   VAR_OUTPUT 
      error { ExternalAccessible := 'False'; ExternalVisible := 'False'; ExternalWritable := 'False'} : Bool;
      status { ExternalAccessible := 'False'; ExternalVisible := 'False'; ExternalWritable := 'False'} : Word;
   END_VAR

   VAR 
      statActorType { ExternalAccessible := 'False'; ExternalVisible := 'False'; ExternalWritable := 'False'} : DInt;
      statByteOffset { ExternalAccessible := 'False'; ExternalVisible := 'False'; ExternalWritable := 'False'} : Int;
      statFirstCycle { ExternalAccessible := 'False'; ExternalVisible := 'False'; ExternalWritable := 'False'} : Bool := TRUE;
      statAddressOut { ExternalAccessible := 'False'; ExternalVisible := 'False'; ExternalWritable := 'False'} : Struct
         RID { ExternalAccessible := 'False'; ExternalVisible := 'False'; ExternalWritable := 'False'} : DWord;
         AREA { ExternalAccessible := 'False'; ExternalVisible := 'False'; ExternalWritable := 'False'} : Byte;
         DB_NUMBER { ExternalAccessible := 'False'; ExternalVisible := 'False'; ExternalWritable := 'False'} : UInt;
         OFFSET { ExternalAccessible := 'False'; ExternalVisible := 'False'; ExternalWritable := 'False'} : UDInt;
      END_STRUCT;
      statNsoll { ExternalAccessible := 'False'; ExternalVisible := 'False'; ExternalWritable := 'False'} : DInt;
      statOutput { ExternalAccessible := 'False'; ExternalVisible := 'False'; ExternalWritable := 'False'} : Int;
   END_VAR

   VAR_TEMP 
      tempAttributes : Byte;
      tempDBLength : UDInt;
      tempStatus : Int;
      tempEno : Bool;
   END_VAR

   VAR CONSTANT 
      AREA_DB : Byte := 16#8B;
      STATUS_DONE : Word := 16#0000;
      STATUS_BUSY : Word := 16#7001;
      ALARM_OPTIMIZED_DB : UDInt := 9106;
      ALARM_INTERNAL : UDInt := 9201;
      ALARM_WRITE_OUTPUT : UDInt := 9401;
   END_VAR


BEGIN
	//================================================================================
	//SIEMENS AG // (c)Copyright 2019 All Rights Reserved
	//--------------------------------------------------------------------------------
	//Library:       LSimaHydTO
	//Tested with:   S7-15xx
	//Engineering:   TIA Portal  V15
	//Restrictions:  -
	//Requirements:  S7-1500 (FW 2.5)
	//Functionality: - for internal use
	//
	//--------------------------------------------------------------------------------
	//Change log table:
	//
	//Version     Date          Expert in charge    Changes applied
	//01.00.00    15.03.2018    APC_ERLF            First released version
	//================================================================================
	// Set error FALSE
	#error := FALSE;
	
	IF (#statFirstCycle)
	THEN
	  // Get adresses from TO
	  #statActorType := #axis.Actor.Type;
	  #statAddressOut.AREA := #axis.Actor.Interface.AddressOut.AREA;
	  #statAddressOut.DB_NUMBER := #axis.Actor.Interface.AddressOut.DB_NUMBER;
	  #statAddressOut.OFFSET := #axis.Actor.Interface.AddressOut.OFFSET;
	  #statAddressOut.RID := #axis.Actor.Interface.AddressOut.RID;
	  
	  IF #statActorType = 0 THEN
	    // analog
	    
	    #statByteOffset := UDINT_TO_INT(#statAddressOut.OFFSET / 8);
	  ELSIF #statActorType = 1 THEN
	    //profidrive
	    #statByteOffset := UDINT_TO_INT(#statAddressOut.OFFSET / 8) + 2;
	  END_IF;
	  
	  IF (#statAddressOut.AREA = #AREA_DB) THEN
	    #tempStatus := ATTR_DB(REQ := TRUE
	                           , DB_NUMBER := #statAddressOut.DB_NUMBER
	                           , DB_LENGTH => #tempDBLength
	                           , ATTRIB => #tempAttributes);
	    
	    IF (#tempStatus <> 0) THEN
	      // Error in reading block data
	      #error := TRUE;
	      #status := UDINT_TO_WORD(#ALARM_INTERNAL);
	      RETURN;
	      
	    ELSIF ((#tempDBLength = 0)
	      AND (#tempAttributes.%X0 = FALSE))
	    THEN
	      // Block is optimized
	      #error := TRUE;
	      #status := UDINT_TO_WORD(#ALARM_OPTIMIZED_DB);
	      RETURN;
	      
	    END_IF;
	  END_IF;
	  
	  #statFirstCycle := FALSE;
	END_IF;
	
	
	#status := #STATUS_BUSY;
	CASE #statActorType OF
	  0: // analog
	    #statOutput := LREAL_TO_INT(0.01 * #setpoint * 27648);
	    POKE(area := #statAddressOut.AREA,
	         dbNumber := #statAddressOut.DB_NUMBER,
	         byteOffset := #statByteOffset,
	         value := INT_TO_WORD(#statOutput),
	         ENO => #tempEno);
	  1: // profidrive
	    #statNsoll := LREAL_TO_DINT(LIMIT(MN := -2.0, IN := 0.01 * #setpoint, MX := 1.999999999) * 1073741824.0);
	    POKE(area := #statAddressOut.AREA,
	         dbNumber := #statAddressOut.DB_NUMBER,
	         byteOffset := #statByteOffset,
	         value := DINT_TO_DWORD(#statNsoll),
	         ENO => #tempEno);
	END_CASE;
	
	
	// Check if read worked
	IF (#tempEno = FALSE) THEN
	  #error := TRUE;
	  
	  #status := UDINT_TO_WORD(#ALARM_WRITE_OUTPUT);
	END_IF;
	
	
	
END_FUNCTION_BLOCK

FUNCTION "LSimaHydTO_GetUnitsCorrection" : LReal
{ S7_Optimized_Access := 'TRUE' }
AUTHOR : APC_ERLF
FAMILY : LSimaHydTO
VERSION : 1.0
   VAR_INPUT 
      lengthUnit : UDInt;
      velocityUnit : UDInt;
   END_VAR

   VAR_OUTPUT 
      accelFactor : LReal;
   END_VAR

   VAR_TEMP 
      tempLengthFactor : LReal;
      tempTimeFactor : LReal;
   END_VAR


BEGIN
	//================================================================================
	//SIEMENS AG // (c)Copyright 2019 All Rights Reserved
	//--------------------------------------------------------------------------------
	//Library:       LSimaHydTO
	//Tested with:   S7-15xx
	//Engineering:   TIA Portal  V15
	//Restrictions:  -
	//Requirements:  S7-1500 (FW 2.5)
	//Functionality: - for internal use
	//
	//--------------------------------------------------------------------------------
	//Change log table:
	//
	//Version     Date          Expert in charge    Changes applied
	//01.00.00    24.04.2020    APC_ERLF            First released version
	//================================================================================
	//
	
	CASE #lengthUnit OF
	    1013: //    mm
	        // get time factor
	        CASE #velocityUnit OF
	            1061, 1062: // m/s, mm/s
	                #tempTimeFactor := 1.0;
	            1524, 1525, 1527:    // mm/min, m/min, km/min
	                #tempTimeFactor := 60.0;
	            1063, 1526, 1064:    // m/h, mm/h, km/h
	                #tempTimeFactor := 3600.0;
	            ELSE
	                #tempTimeFactor := 1.0;
	        END_CASE;
	        // get length factor
	        CASE #velocityUnit OF
	            1062, 1524, 1526:  // mm/s, mm/min, mm/h
	                #tempLengthFactor := 1.0;
	                #accelFactor := 1.0;
	            1061, 1525, 1063:  // m/s, m/min, m/h
	                #tempLengthFactor := 1000.0;
	                #accelFactor := 0.001;
	            1064, 1527: //   km/h, km/min
	                #tempLengthFactor := 1000000.0;
	                #accelFactor := 0.001;
	            ELSE
	                #tempLengthFactor := 1.0;
	                #accelFactor := 1.0;
	        END_CASE;
	        
	    1019: //    in
	        // get time factor
	        CASE #velocityUnit OF
	            1066, 1067: // in/s, ft/s
	                #tempTimeFactor := 1.0;
	            1069, 1070: // in/min, ft/min
	                #tempTimeFactor := 60.0;
	            1075:       // mi/h
	                #tempTimeFactor := 3600.0;
	            ELSE
	                #tempTimeFactor := 1.0;
	        END_CASE;
	        // get length factor
	        CASE #velocityUnit OF
	            1066, 1069:  // in/s, in/min
	                #tempLengthFactor := 1.0;
	                #accelFactor := 1.0;
	            1067, 1070:  // ft/s, ft/min
	                #tempLengthFactor := 12.0;
	                #accelFactor := 1.0/#tempLengthFactor;
	            1075:       // mi/h
	                #tempLengthFactor := 63360.0;
	                #accelFactor := 1.0 / 12.0;
	            ELSE
	                #tempLengthFactor := 1.0;
	                #accelFactor := 1.0;
	        END_CASE;
	        
	        
	    1010: //    m
	        // get time factor
	        CASE #velocityUnit OF
	            1061, 1062: // m/s, mm/s
	                #tempTimeFactor := 1.0;
	            1524, 1525, 1527:    // mm/min, m/min, km/min
	                #tempTimeFactor := 60.0;
	            1063, 1526, 1064:    // m/h, mm/h, km/h
	                #tempTimeFactor := 3600.0;
	            ELSE
	                #tempTimeFactor := 1.0;
	        END_CASE;
	        // get length factor
	        CASE #velocityUnit OF
	            1062, 1524, 1526:  // mm/s, mm/min, mm/h
	                #tempLengthFactor := 0.001;
	                #accelFactor := 1000.0;
	            1061, 1525, 1063:  // m/s, m/min, m/h
	                #tempLengthFactor := 1.0;
	                #accelFactor := 1.0;
	            1064, 1527: //   km/h, km/min
	                #tempLengthFactor := 1000.0;
	                #accelFactor := 1.0;
	            ELSE
	                #tempLengthFactor := 1.0;
	                #accelFactor := 1.0;
	        END_CASE;
	        
	    1018: //    ft
	        // get time factor
	        CASE #velocityUnit OF
	            1066, 1067: // in/s, ft/s
	                #tempTimeFactor := 1.0;
	            1069, 1070: // in/min, ft/min
	                #tempTimeFactor := 60.0;
	            1075:       // mi/h
	                #tempTimeFactor := 3600.0;
	            ELSE
	                #tempTimeFactor := 1.0;
	        END_CASE;
	        // get length factor
	        CASE #velocityUnit OF
	            1066, 1069:  // in/s, in/min
	                #tempLengthFactor := 0.0833333;
	                #accelFactor := 12.0;
	            1067, 1070:  // ft/s, ft/min
	                #tempLengthFactor := 1.0;
	                #accelFactor := 1.0;
	            1075:       // mi/h
	                #tempLengthFactor := 5280.0;
	                #accelFactor := 1.0;
	            ELSE
	                #tempLengthFactor := 1.0;
	                #accelFactor := 1.0;
	        END_CASE;
	    1005, 1004: //    °,rad 
	        // get time factor
	        CASE #velocityUnit OF
	            1086, 1521: // rad/s,°/s 
	                #tempTimeFactor := 1.0;
	            1522, 1523: // °/min, rad/min
	                #tempTimeFactor := 60.0;
	            ELSE
	                #tempTimeFactor := 1.0;
	        END_CASE;
	        #tempLengthFactor := 1.0;
	        #accelFactor := 1.0;
	    1014: //    µm
	        // get time factor
	        CASE #velocityUnit OF
	            1061, 1062: // m/s, mm/s
	                #tempTimeFactor := 1.0;
	            1524, 1525, 1527:    // mm/min, m/min, km/min
	                #tempTimeFactor := 60.0;
	            1063, 1526, 1064:    // m/h, mm/h, km/h
	                #tempTimeFactor := 3600.0;
	            ELSE
	                #tempTimeFactor := 1.0;
	        END_CASE;
	        // get length factor
	        CASE #velocityUnit OF
	            1062, 1524, 1526:  // mm/s, mm/min, mm/h
	                #tempLengthFactor := 1.0E+3;
	                #accelFactor := 1.0E-3;
	            1061, 1525, 1063:  // m/s, m/min, m/h
	                #tempLengthFactor := 1.0E+6;
	                #accelFactor := 1.0E-6;
	            1064, 1527: //   km/h, km/min
	                #tempLengthFactor := 1.0E+9;
	                #accelFactor := 1.0E-6;
	            ELSE
	                #tempLengthFactor := 1.0;
	                #accelFactor := 1.0;
	        END_CASE;
	        
	    1015: //    nm
	        // get time factor
	        CASE #velocityUnit OF
	            1061, 1062: // m/s, mm/s
	                #tempTimeFactor := 1.0;
	            1524, 1525, 1527:    // mm/min, m/min, km/min
	                #tempTimeFactor := 60.0;
	            1063, 1526, 1064:    // m/h, mm/h, km/h
	                #tempTimeFactor := 3600.0;
	            ELSE
	                #tempTimeFactor := 1.0;
	        END_CASE;
	        // get length factor
	        CASE #velocityUnit OF
	            1062, 1524, 1526:  // mm/s, mm/min, mm/h
	                #tempLengthFactor := 1.0E+6;
	                #accelFactor := 1.0E-6;
	            1061, 1525, 1063:  // m/s, m/min, m/h
	                #tempLengthFactor := 1.0E+9;
	                #accelFactor := 1.0E-9;
	            1064, 1527: //   km/h, km/min
	                #tempLengthFactor := 1.0E+12;
	                #accelFactor := 1.0E-9;
	            ELSE
	                #tempLengthFactor := 1.0;
	                #accelFactor := 1.0;
	        END_CASE;
	        
	    1011: //    km
	        // get time factor
	        CASE #velocityUnit OF
	            1061, 1062: // m/s, mm/s
	                #tempTimeFactor := 1.0;
	            1524, 1525, 1527:    // mm/min, m/min, km/min
	                #tempTimeFactor := 60.0;
	            1063, 1526, 1064:    // m/h, mm/h, km/h
	                #tempTimeFactor := 3600.0;
	            ELSE
	                #tempTimeFactor := 1.0;
	        END_CASE;
	        // get length factor
	        CASE #velocityUnit OF
	            1062, 1524, 1526:  // mm/s, mm/min, mm/h
	                #tempLengthFactor := 1.0E-6;
	                #accelFactor := 1.0E+6;
	            1061, 1525, 1063:  // m/s, m/min, m/h
	                #tempLengthFactor := 1.0E-3;
	                #accelFactor := 1.0E+3;
	            1064, 1527: //   km/h, km/min
	                #tempLengthFactor := 1.0;
	                #accelFactor := 1.0E+3;
	            ELSE
	                #tempLengthFactor := 1.0;
	                #accelFactor := 1.0;
	        END_CASE;
	        
	    1021: //    mi
	        // get time factor
	        CASE #velocityUnit OF
	            1066, 1067: // in/s, ft/s
	                #tempTimeFactor := 1.0;
	            1069, 1070: // in/min, ft/min
	                #tempTimeFactor := 60.0;
	            1075:       // mi/h
	                #tempTimeFactor := 3600.0;
	            ELSE
	                #tempTimeFactor := 1.0;
	        END_CASE;
	        // get length factor
	        CASE #velocityUnit OF
	            1066, 1069:  // in/s, in/min
	                #tempLengthFactor := 1.0 / 63360.0;
	                #accelFactor := 63360.0;
	            1067, 1070:  // ft/s, ft/min
	                #tempLengthFactor := 1.0 / 5280.0;
	                #accelFactor := 5280.0;
	            1075:       // mi/h
	                #tempLengthFactor := 1.0;
	            ELSE
	                #tempLengthFactor := 1.0;
	                #accelFactor := 1.0;
	        END_CASE;
	        
	    ELSE
	        #tempTimeFactor := 1.0;
	        #tempLengthFactor := 1.0;
	        #accelFactor := 1.0;
	END_CASE;
	
	#LSimaHydTO_GetUnitsCorrection := #tempTimeFactor / #tempLengthFactor;
END_FUNCTION

FUNCTION "LSimaHydTO_Transducer" : Void
{ S7_Optimized_Access := 'TRUE' }
AUTHOR : APC_ERLF
FAMILY : LSimaHydTO
VERSION : 1.0
   VAR_INPUT 
      rawValue : Word;
      forceFactor : LReal;
   END_VAR

   VAR_IN_OUT 
      statusTransducer : "LSimaHydTO_typeStatusTransducer";
      transducer : "LSimaHydTO_typeTransducer";
   END_VAR


BEGIN
	//================================================================================
	//SIEMENS AG // (c)Copyright 2019 All Rights Reserved
	//--------------------------------------------------------------------------------
	//Library:       LSimaHydTO
	//Tested with:   S7-15xx
	//Engineering:   TIA Portal  V15
	//Restrictions:  -
	//Requirements:  S7-1500 (FW 2.5)
	//Functionality: - for internal use
	//
	//--------------------------------------------------------------------------------
	//Change log table:
	//
	//Version     Date          Expert in charge    Changes applied
	//01.00.00    15.03.2018    APC_ERLF            First released version
	//================================================================================
	
	#statusTransducer.RawValue := #rawValue;
	IF #transducer.ErrorValue = #statusTransducer.RawValue THEN
	  #statusTransducer.Error := TRUE;
	ELSE
	  #statusTransducer.PressureValue := WORD_TO_INT(#statusTransducer.RawValue) * #transducer.NominalPressure /
	  INT_TO_REAL(#transducer.HWReference) + #transducer.Offset;
	  #statusTransducer.ForceValue := #statusTransducer.PressureValue * #transducer.Area * #forceFactor;
	  #statusTransducer.Error := FALSE;
	END_IF;
	
	
END_FUNCTION

FUNCTION "LSimaHydTO_Profile" : LReal
{ S7_Optimized_Access := 'TRUE' }
AUTHOR : APC_ERLF
FAMILY : LSimaHydTO
VERSION : 1.0
   VAR_INPUT 
      inputValue : LReal;
   END_VAR

   VAR_OUTPUT 
      inProfile : Bool;
   END_VAR

   VAR_IN_OUT 
      profile : "LSimaHydTO_typeProfile";
   END_VAR

   VAR_TEMP 
      tempSetPoint : LReal;
      tempV0 : LReal;
      tempV1 : LReal;
      tempQ0 : LReal;
      tempQ1 : LReal;
      tempRetValue : LReal;
      tempIdx : DInt;
      tempBegIdx : DInt;
      tempEndIdx : DInt;
      tempMinValue : LReal;
      tempMaxValue : LReal;
   END_VAR


BEGIN
	//================================================================================
	//SIEMENS AG // (c)Copyright 2019 All Rights Reserved
	//--------------------------------------------------------------------------------
	//Library:       LSimaHydTO
	//Tested with:   S7-15xx
	//Engineering:   TIA Portal  V15
	//Restrictions:  -
	//Requirements:  S7-1500 (FW 2.5)
	//Functionality: - for internal use
	//
	//--------------------------------------------------------------------------------
	//Change log table:
	//
	//Version     Date          Expert in charge    Changes applied
	//01.00.00    15.03.2018    APC_ERLF            First released version
	//================================================================================
	
	#tempBegIdx := 0;
	#tempEndIdx := LIMIT(MN := 0,IN := #profile.MaxIdx,MX := "LSIMAHYD_PROFILE_POINTS_UPPER_LIMIT");
	#tempMinValue := #profile.LeadingValue[#tempBegIdx];
	#tempMaxValue := #profile.LeadingValue[#tempEndIdx];
	#inProfile := #inputValue >= #tempMinValue AND #inputValue <= #tempMaxValue;
	#tempSetPoint := LIMIT(MN := #tempMinValue, IN := (#inputValue), MX := #tempMaxValue);
	WHILE (#tempEndIdx - #tempBegIdx) >= 2 DO
	  #tempIdx := (#tempEndIdx + #tempBegIdx) / 2;
	  IF (#profile.LeadingValue[#tempIdx] >= #tempSetPoint )
	  THEN
	    #tempEndIdx := #tempIdx;
	  ELSE
	    #tempBegIdx := #tempIdx;
	  END_IF;
	END_WHILE;
	#tempV0 := #profile.LeadingValue[#tempBegIdx];
	#tempV1 := #profile.LeadingValue[#tempEndIdx];
	#tempQ0 := #profile.Value[#tempBegIdx];
	#tempQ1 := #profile.Value[#tempEndIdx];
	IF #tempV0 = #tempV1 THEN
	  #tempRetValue := (#tempQ0 + #tempQ1) / 2.0;
	ELSE
	  #tempRetValue := #tempQ0 + (#tempQ1 - #tempQ0) * (#tempSetPoint - #tempV0) / (#tempV1 - #tempV0);
	END_IF;
	#LSimaHydTO_Profile :=  #tempRetValue;
	
	
END_FUNCTION

FUNCTION "LSimaHydTO_Internal_1" : Void
{ S7_Optimized_Access := 'TRUE' }
AUTHOR : APC_ERLF
FAMILY : LSimaHydTO
VERSION : 1.0
   VAR_IN_OUT 
      "var" : Variant;
   END_VAR

   VAR_TEMP 
      tempVar : "LSimaHydTO_typeVCharData";
      tempProf : "LSimaHydTO_typeProfile";
      tempAxisData : "LSimaHydTO_typeAxisData";
   END_VAR


BEGIN
	//================================================================================
	//SIEMENS AG // (c)Copyright 2019 All Rights Reserved
	//--------------------------------------------------------------------------------
	//Library:       LSimaHydTO
	//Tested with:   S7-15xx
	//Engineering:   TIA Portal  V15
	//Restrictions:  -
	//Requirements:  S7-1500 (FW 2.5)
	//Functionality: - for internal use
	//
	//--------------------------------------------------------------------------------
	//Change log table:
	//
	//Version     Date          Expert in charge    Changes applied
	//01.00.00    15.03.2018    APC_ERLF            First released version
	//================================================================================
	
	
	"LSimaHydTO_Internal_2"(#tempVar);
	"LSimaHydTO_Internal_2"(#tempProf);
	"LSimaHydTO_Internal_2"(#tempAxisData);
	
	
	
END_FUNCTION

FUNCTION "LSimaHydTO_Internal_2" : Void
{ S7_Optimized_Access := 'TRUE' }
AUTHOR : APC_ERLF
FAMILY : LSimaHydTO
VERSION : 1.0
   VAR_IN_OUT 
      "var" : Variant;
   END_VAR


BEGIN
	//================================================================================
	//SIEMENS AG // (c)Copyright 2019 All Rights Reserved
	//--------------------------------------------------------------------------------
	//Library:       LSimaHydTO
	//Tested with:   S7-15xx
	//Engineering:   TIA Portal  V15
	//Restrictions:  -
	//Requirements:  S7-1500 (FW 2.5)
	//Functionality: - for internal use
	//
	//--------------------------------------------------------------------------------
	//Change log table:
	//
	//Version     Date          Expert in charge    Changes applied
	//01.00.00    15.03.2018    APC_ERLF            First released version
	//================================================================================
	
	
	
END_FUNCTION

FUNCTION "LSimaHydTO_RampGen" : Void
{ S7_Optimized_Access := 'TRUE' }
AUTHOR : APC_ERLF
FAMILY : LSimaHydTO
VERSION : 1.0
   VAR_INPUT 
      inputValue : LReal;
      acceleration : LReal;
      deceleration : LReal;
      sampleTime : LReal;
   END_VAR

   VAR_OUTPUT 
      active : Bool;
   END_VAR

   VAR_IN_OUT 
      outputValue : LReal;
   END_VAR

   VAR_TEMP 
      tempUpNullStep : LReal;
      tempStepUp : LReal;
      tempStepDown : LReal;
      tempAuxOutput : LReal;
      tempAuxStep : LReal;
   END_VAR


BEGIN
	//================================================================================
	//SIEMENS AG // (c)Copyright 2019 All Rights Reserved
	//--------------------------------------------------------------------------------
	//Library:       LSimaHydTO
	//Tested with:   S7-15xx
	//Engineering:   TIA Portal  V15
	//Restrictions:  -
	//Requirements:  S7-1500 (FW 2.5)
	//Functionality: - for internal use
	//
	//--------------------------------------------------------------------------------
	//Change log table:
	//
	//Version     Date          Expert in charge    Changes applied
	//01.00.00    15.03.2018    APC_ERLF            First released version
	//================================================================================
	
	#tempStepUp := #acceleration * #sampleTime;
	#tempStepDown := #deceleration * #sampleTime;
	#tempAuxOutput := #outputValue;
	IF #inputValue >= 0.0 AND #tempAuxOutput < 0.0 OR
	  #inputValue <= 0.0 AND #tempAuxOutput > 0.0 THEN  // bigger as 0 
	  IF ABS(#tempAuxOutput) >= #tempStepDown THEN
	    IF #tempAuxOutput > 0 THEN  //positive
	      #tempAuxOutput := #tempAuxOutput - #tempStepDown;
	    ELSE  //negative
	      #tempAuxOutput := #tempAuxOutput + #tempStepDown;
	    END_IF;
	    #active := TRUE;
	  ELSE
	    #tempUpNullStep := #tempStepUp * (1 - ABS(#tempAuxOutput) / #tempStepDown);
	    IF ABS(#inputValue) > #tempUpNullStep THEN  //RG active
	      IF #inputValue > 0 THEN  //positive
	        #tempAuxOutput := #tempUpNullStep;
	      ELSE  //negative
	        #tempAuxOutput := - #tempUpNullStep;
	      END_IF;
	      #active := TRUE;
	    ELSE
	      #tempAuxOutput := #inputValue;
	      #active := FALSE;
	    END_IF;
	  END_IF;
	ELSE
	  IF ABS(#inputValue) > ABS(#tempAuxOutput) THEN  //up
	    #tempAuxStep := #tempStepUp;
	  ELSE
	    #tempAuxStep := - #tempStepDown;
	  END_IF;
	  IF ABS(#inputValue - #tempAuxOutput) > ABS(#tempAuxStep) THEN  //RG active
	    IF #inputValue > 0 THEN  //positive
	      #tempAuxOutput := #tempAuxOutput + #tempAuxStep;
	    ELSE  //negative
	      #tempAuxOutput := #tempAuxOutput - #tempAuxStep;
	    END_IF;
	    #active := TRUE;
	  ELSE  //RG inactive
	    #tempAuxOutput := #inputValue;
	    #active := FALSE;
	  END_IF;
	END_IF;
	#outputValue := #tempAuxOutput;
END_FUNCTION

FUNCTION "LSimaHydTO_Vchar" : LReal
{ S7_Optimized_Access := 'TRUE' }
AUTHOR : APC_ERLF
FAMILY : LSimaHydTO
VERSION : 1.0
   VAR_INPUT 
      VChar : REF_TO "LSimaHydTO_typeVCharData";
      setPoint : LReal;
      qOutput : LReal;
      forward : Bool;
      backward : Bool;
   END_VAR

   VAR_TEMP 
      tempSetPoint : LReal;
      tempV0 : LReal;
      tempV1 : LReal;
      tempQ0 : LReal;
      tempQ1 : LReal;
      tempRetValue : LReal;
      tempIdx : DInt;
      tempBegIdx : DInt;
      tempEndIdx : DInt;
      tempInverse : Bool;
      tempZeroZonePos : LReal;
      tempZeroZoneNeg : LReal;
   END_VAR


BEGIN
	//================================================================================
	//SIEMENS AG // (c)Copyright 2019 All Rights Reserved
	//--------------------------------------------------------------------------------
	//Library:       LSimaHydTO
	//Tested with:   S7-15xx
	//Engineering:   TIA Portal  V15
	//Restrictions:  -
	//Requirements:  S7-1500 (FW 2.5)
	//Functionality: - for internal use
	//
	//--------------------------------------------------------------------------------
	//Change log table:
	//
	//Version     Date          Expert in charge    Changes applied
	//01.00.00    15.03.2018    APC_ERLF            First released version
	//================================================================================
	
	#tempSetPoint := LIMIT(MN := #VChar^.VelocityLimitNegative, IN := (#setPoint), MX := #VChar^.VelocityLimitPositive);
	#tempBegIdx := 0;
	#tempEndIdx := #VChar^.MaxIdx;
	
	#tempInverse := #VChar^.Velocity[#tempEndIdx] < #VChar^.Velocity[#tempBegIdx];
	WHILE (#tempEndIdx - #tempBegIdx) >= 2 DO
	  #tempIdx := (#tempEndIdx + #tempBegIdx) / 2;
	  IF (#VChar^.Velocity[#tempIdx] >= #tempSetPoint AND NOT #tempInverse)
	    OR
	    (#VChar^.Velocity[#tempIdx] <= #tempSetPoint AND #tempInverse)
	  THEN
	    #tempEndIdx := #tempIdx;
	  ELSE
	    #tempBegIdx := #tempIdx;
	  END_IF;
	END_WHILE;
	
	#tempV0 := #VChar^.Velocity[#tempBegIdx];
	#tempV1 := #VChar^.Velocity[#tempEndIdx];
	#tempQ0 := #VChar^.QOutput[#tempBegIdx];
	#tempQ1 := #VChar^.QOutput[#tempEndIdx];
	
	IF #tempV0 = #tempV1 THEN
	  #tempRetValue := (#tempQ0 + #tempQ1) / 2.0;
	ELSE
	  #tempRetValue := #tempQ0 + (#tempQ1 - #tempQ0) * (#tempSetPoint - #tempV0) / (#tempV1 - #tempV0);
	END_IF;
	
	// new 
	IF #VChar^.ZeroZonePositive <> 0.0
	  AND #VChar^.ZeroZoneNegative <> 0.0
	THEN
	  #tempZeroZoneNeg := - ABS(#VChar^.ZeroZoneNegative);
	  #tempZeroZonePos := ABS(#VChar^.ZeroZonePositive);
	  IF #tempRetValue <= #tempZeroZonePos
	    AND #tempRetValue >= #tempZeroZoneNeg
	  THEN
	    IF #forward OR #qOutput >= #tempZeroZonePos THEN
	      #tempRetValue := #tempZeroZonePos;
	    ELSIF #backward OR #qOutput <= #tempZeroZoneNeg THEN
	      #tempRetValue := #tempZeroZoneNeg;
	    ELSE
	      #tempRetValue := 0.5 * (#tempZeroZonePos + #tempZeroZoneNeg);
	    END_IF;
	    IF NOT (#forward OR #backward) AND #setPoint = 0.0 THEN
	      #tempRetValue := 0.5 * (#tempZeroZonePos + #tempZeroZoneNeg);
	    END_IF;
	    
	    
	  END_IF;
	END_IF;
	#LSimaHydTO_Vchar := LIMIT(MN := #VChar^.QOutput[0], IN := #tempRetValue, MX := #VChar^.QOutput[#VChar^.MaxIdx]);
	
END_FUNCTION

FUNCTION "LSimaHydTO_Scale" : LReal
{ S7_Optimized_Access := 'TRUE' }
AUTHOR : APC_ERLF
FAMILY : LSimaHydTO
VERSION : 1.0
   VAR_INPUT 
      input : LReal;
      inBegin : LReal;
      inEnd : LReal;
      valBegin : LReal;
      valEnd : LReal;
   END_VAR

   VAR_TEMP 
      tempOut : LReal;
   END_VAR


BEGIN
	//================================================================================
	//SIEMENS AG // (c)Copyright 2019 All Rights Reserved
	//--------------------------------------------------------------------------------
	//Library:       LSimaHydTO
	//Tested with:   S7-15xx
	//Engineering:   TIA Portal  V15
	//Restrictions:  -
	//Requirements:  S7-1500 (FW 2.5)
	//Functionality: - for internal use
	//
	//--------------------------------------------------------------------------------
	//Change log table:
	//
	//Version     Date          Expert in charge    Changes applied
	//01.00.00    15.03.2018    APC_ERLF            First released version
	//================================================================================
	
	
	// Function scales output value dependent upon the input value
	// 
	// Use the "FC_BC_Scale" instruction to scale a floating-point number by mapping it to a specific value range.
	// You specify the value range with the valBegin and valEnd parameters. The result of the scaling is an Lreal.
	//
	// The following figure shows an example of how values can be scaled:
	//
	//
	//   valEnd |               _______________
	//          |              /|
	//          |             / |
	//          |            /  |
	// valBegin |___________/   |
	//          |___________|___|______________________________________
	//               inBegin     inEnd
	//               
	//
	
	
	IF #inEnd <= #inBegin THEN
	  #tempOut := 1.0;
	ELSIF #input <= #inBegin THEN
	  #tempOut := #valBegin;
	ELSIF #input > #inBegin AND #input < #inEnd THEN
	  #tempOut := #valBegin + (#input - #inBegin) * (#valEnd - #valBegin) / (#inEnd - #inBegin);
	ELSIF #input >= #inEnd THEN
	  #tempOut := #valEnd;
	ELSE
	  #tempOut := 1.0;
	END_IF;
	#LSimaHydTO_Scale := #tempOut;
	
	
END_FUNCTION

FUNCTION "LSimaHydTO_VcharInverse" : LReal
{ S7_Optimized_Access := 'TRUE' }
AUTHOR : APC_ERLF
FAMILY : LSimaHydTO
VERSION : 1.0
   VAR_INPUT 
      qOutput : LReal;
   END_VAR

   VAR_IN_OUT 
      VChar : "LSimaHydTO_typeVCharData";
   END_VAR

   VAR_TEMP 
      tempQOutput : LReal;
      tempV0 : LReal;
      tempV1 : LReal;
      tempQ0 : LReal;
      tempQ1 : LReal;
      tempIdx : DInt;
      tempBegIdx : DInt;
      tempEndIdx : DInt;
      tempRetValue : LReal;
   END_VAR


BEGIN
	//================================================================================
	//SIEMENS AG // (c)Copyright 2019 All Rights Reserved
	//--------------------------------------------------------------------------------
	//Library:       LSimaHydTO
	//Tested with:   S7-15xx
	//Engineering:   TIA Portal  V15
	//Restrictions:  -
	//Requirements:  S7-1500 (FW 2.5)
	//Functionality: - for internal use
	//
	//--------------------------------------------------------------------------------
	//Change log table:
	//
	//Version     Date          Expert in charge    Changes applied
	//01.00.00    15.03.2018    APC_ERLF            First released version
	//================================================================================
	
	
	#tempBegIdx := 0;
	#tempEndIdx := #VChar.MaxIdx;
	#tempQOutput := LIMIT(MN := #VChar.QOutput[#tempBegIdx], IN := #qOutput, MX := #VChar.QOutput[#tempEndIdx]);
	IF (#tempQOutput) < #VChar.ZeroZonePositive
	  AND
	  (#tempQOutput) > - ABS(#VChar.ZeroZoneNegative)
	THEN
	  #tempRetValue := 0.0;
	ELSE
	  WHILE (#tempEndIdx - #tempBegIdx) >= 2 DO
	    #tempIdx := (#tempEndIdx + #tempBegIdx) / 2;
	    IF (#VChar.QOutput[#tempIdx] >= #tempQOutput)
	    THEN
	      #tempEndIdx := #tempIdx;
	    ELSE
	      #tempBegIdx := #tempIdx;
	    END_IF;
	  END_WHILE;
	  #tempV0 := #VChar.Velocity[#tempBegIdx];
	  #tempV1 := #VChar.Velocity[#tempEndIdx];
	  #tempQ0 := #VChar.QOutput[#tempBegIdx];
	  #tempQ1 := #VChar.QOutput[#tempEndIdx];
	  IF #tempQ0 = #tempQ1 THEN
	    #tempRetValue := (#tempV0 + #tempV1) / 2.0;
	  ELSE
	    #tempRetValue := #tempV0 + (#tempV1 - #tempV0) * (#tempQOutput - #tempQ0) / (#tempQ1 - #tempQ0);
	  END_IF;
	END_IF;
	#LSimaHydTO_VcharInverse := #tempRetValue; 
	
	
END_FUNCTION

FUNCTION_BLOCK "LSimaHydTO_HydSyncAxis"
{ S7_Optimized_Access := 'TRUE' }
AUTHOR : APC_ERLF
FAMILY : LSimaHydTO
VERSION : 1.0
   VAR_IN_OUT 
      axisTO {InstructionName := 'TO_SynchronousAxis'; LibVersion := '4.0'} : TO_SynchronousAxis;
      axisData : "LSimaHydTO_typeAxisData";
      instHydAxisFB : "LSimaHydTO_HydAxis";
   END_VAR


BEGIN
	//================================================================================
	//SIEMENS AG // (c)Copyright 2019 All Rights Reserved
	//--------------------------------------------------------------------------------
	//Library:       LSimaHydTO
	//Tested with:   S7-15xx
	//Engineering:   TIA Portal  V15
	//Restrictions:  -
	//Requirements:  S7-1500 (FW 2.5)
	//Functionality: - for internal use
	//
	//--------------------------------------------------------------------------------
	//Change log table:
	//
	//Version     Date          Expert in charge    Changes applied
	//01.00.00    15.03.2018    APC_ERLF            First released version
	//================================================================================
	
	//Call function block
	#instHydAxisFB(axisTO := #axisTO,
	                   axisData := #axisData);
	
END_FUNCTION_BLOCK

FUNCTION_BLOCK "SimaHydTO_AxisBasics_PosAxis"   // FB33191, FBD
TITLE = SimaHydTO_AxisBasics_PosAxis
{ S7_Optimized_Access := 'TRUE' }
FAMILY : SimaHydTO/LAxisBasics
VERSION : 1.0
// Function block information: See Function block network 1
// stored: AutoNumber true, IsIECCheckEnabled false, IsRetainMemResEnabled false, MemoryReserve 100, SetENOAutomatically false, UDAEnableTagReadback false
   VAR_INPUT
      axis : TO_PositioningAxis;   // Technology object (axis)
      powerEnable : Bool;   // MC_Power: 0: The technology object is disabled / 1: The technology object is enabled
      powerStartMode : DInt := 1;   // 0: Enable axis not position-controlled / 1: Enable axis position-controlled
      powerStopMode : Int := 0;   // 0: Emergency stop / 1: Immediate stop / 2: Stop with maximum dynamic values
      resetExecute : Bool;   // MC_Reset: Start job with a positive edge
      resetRestart : Bool := false;   // 0: Acknowledgment of queued technology alarms / 1: Reinitialization of the technology object and acknowledgment of pending technology alarms
      homeExecute : Bool;   // MC_Home: Start job with a positive edge
      homePosition : LReal;   // The specified value is used according to the selected "Mode".
      homeMode : Int;   // 0: Direct homing (absolute) / 1: Direct homing (relative) / 2: Passive homing / 3: Active homing / 4: Reserved / 5: Active homing (<TO>.Homing.HomePosition) / 6: Absolute encoder adjustment (relative) / 7: Absolute encoder adjustment (absolute) / 8: Passive homing / 9: Abort passive homing / 10: Passive homing (<TO>.Homing.HomePosition)
      jogForward : Bool;   // MC_MoveJog: As long as the parameter is TRUE, the axis moves in the positive direction
      jogBackward : Bool;   // MC_MoveJog: As long as the parameter is TRUE, the axis moves in the negative direction
      jogVelocity : LReal := 100.0;   // Velocity setpoint / speed setpoint for the motion
      jogAcceleration : LReal := -1.0;   // Acceleration of jog movement
      jogDeceleration : LReal := -1.0;   // Deceleration of jog movement
      jogJerk : LReal := -1.0;   // Jerk of jog movement
      jogPositionControlled : Bool := true;   // 0: Non position-controlled operation / 1: Position-controlled mode - The parameter applies as long as the MC_MoveJog command is executed. After this, the setting of MC_Power applies again.
   END_VAR
   VAR_OUTPUT
      powerStatus { ExternalWritable := 'False'} : Bool;   // MC_Power: 0: Technology object disabled / 1: Technology object enabled
      powerBusy { ExternalWritable := 'False'} : Bool;   // MC_Power: Job is running
      resetDone { ExternalWritable := 'False'} : Bool;   // MC_Reset: Error has been acknowledged or Restart has been executed.
      resetBusy { ExternalWritable := 'False'} : Bool;   // MC_Reset: Job is running
      homeDone { ExternalWritable := 'False'} : Bool;   // MC_Home: Job is completed
      homeBusy { ExternalWritable := 'False'} : Bool;   // MC_Home: Job is running
      jogInVelocity { ExternalWritable := 'False'} : Bool;   // MC_MoveJog: The velocity setpoint / speed setpoint was reached and will be maintained
      jogBusy { ExternalWritable := 'False'} : Bool;   // MC_MoveJog: Job is running
      commandAborted { ExternalWritable := 'False'} : Bool;   // The job was aborted by another job during execution (see also StatusID)
      error { ExternalWritable := 'False'} : Bool;   // An error occurred during execution of the job. The job is rejected. The cause of the error can be found in the "ErrorID" parameter.
      errorID { ExternalWritable := 'False'} : Word;   // ErrorID of motion control instruction (see also StatusID)
      statusID { ExternalWritable := 'False'} : Int;   // Additional specification of affected Motion control instruction of CommandAborted or Error: 0: No instruction / 1: MC_Power / 2: MC_Reset / 3: MC_Home / 4: MC_MoveJog
   END_VAR
   VAR
      instMcPower { ExternalAccessible := 'False'; ExternalVisible := 'False'; ExternalWritable := 'False'; S7_SetPoint := 'True'} : MC_POWER;   // PLCopen functions of basic motion control
      instMcReset { ExternalAccessible := 'False'; ExternalVisible := 'False'; ExternalWritable := 'False'; S7_SetPoint := 'True'} : MC_RESET;
      instMcHome { ExternalAccessible := 'False'; ExternalVisible := 'False'; ExternalWritable := 'False'; S7_SetPoint := 'True'} : MC_HOME;
      instMcMoveJog { ExternalAccessible := 'False'; ExternalVisible := 'False'; ExternalWritable := 'False'; S7_SetPoint := 'True'} : MC_MOVEJOG;
      statCommandAborted { ExternalAccessible := 'False'; ExternalVisible := 'False'; ExternalWritable := 'False'} : Array[#ARRAY_BEGIN..#ARRAY_END] of Bool;   // Arrays to save error information of PLCopen functions
      statError { ExternalAccessible := 'False'; ExternalVisible := 'False'; ExternalWritable := 'False'} : Array[#ARRAY_BEGIN..#ARRAY_END] of Bool;
      statErrorID { ExternalAccessible := 'False'; ExternalVisible := 'False'; ExternalWritable := 'False'} : Array[#ARRAY_BEGIN..#ARRAY_END] of Word;
      MC_MOVEABSOLUTE_Instance { S7_SetPoint := 'True'} : MC_MOVEABSOLUTE;
   END_VAR
   VAR_TEMP
      tempDwordCommandAborted : DWord;   // Variables to check error informations of PLCopen functions
      tempDwordError : DWord;
      tempCount : Int;   // Counter of FOR counting loop
   END_VAR
   VAR CONSTANT
      ARRAY_BEGIN : Int := 1;   // Start-Index of array (Maximum 32 Array elements!)
      ARRAY_END : Int := 32;   // End-Index of array (Maximum 32 Array elements!)
      ERROR_DEFAULT : Bool := false;   // Default values of output signals
      ERRORID_DEFAULT : Word := 16#0;
      STATUSID_DEFAULT : Int := 0;
   END_VAR
BEGIN

REGION Network 1 (SCL): Axis Basics - Header
   //=============================================================================
   //SIEMENS AG
   //(c)Copyright 2016 All Rights Reserved
   //-----------------------------------------------------------------------------
   //Library:       AxisBasics
   //Tested with:   S7-1500 V2.5
   //Engineering:   TIA Portal V15
   //Restrictions:  Motion Control Library V4.0
   //Requirements:  S7-1500(T)
   //Functionality: Basic axis control of TO_PositioningAxis
   //-----------------------------------------------------------------------------
   //Change log table:
   //Version  Date       Expert in charge Changes applied
   //01.00.00 04.10.2018 ArSc             First released version
   //=============================================================================
END_REGION

REGION Network 2: Axis Basics - MC_Power
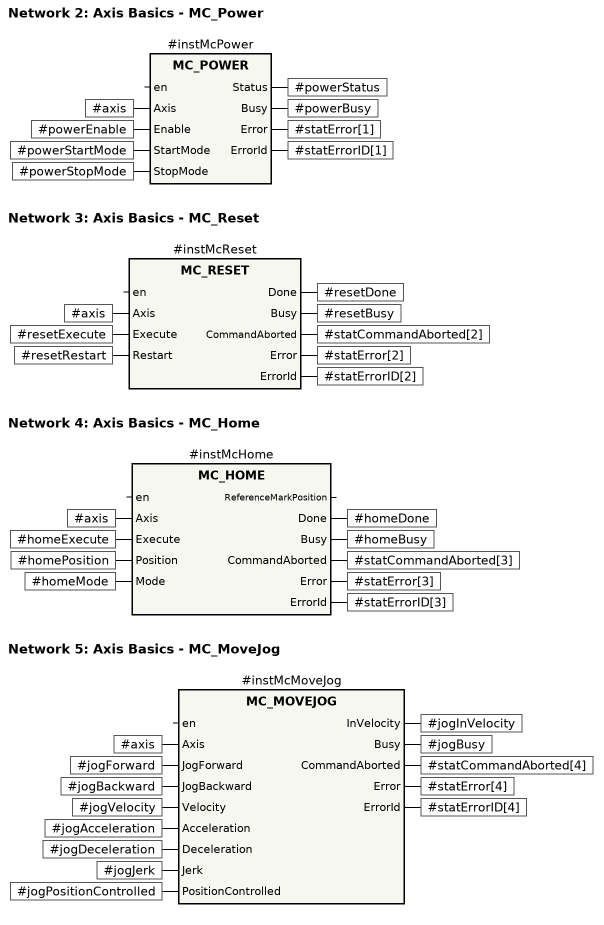
   #instMcPower(Axis := #axis,   // MC_POWER
                Enable := #powerEnable,
                StartMode := #powerStartMode,
                StopMode := #powerStopMode,
                Status => #powerStatus,
                Busy => #powerBusy,
                Error => #statError[1],
                ErrorId => #statErrorID[1]);
END_REGION

REGION Network 3: Axis Basics - MC_Reset
   #instMcReset(Axis := #axis,   // MC_RESET
                Execute := #resetExecute,
                Restart := #resetRestart,
                Done => #resetDone,
                Busy => #resetBusy,
                CommandAborted => #statCommandAborted[2],
                Error => #statError[2],
                ErrorId => #statErrorID[2]);
END_REGION

REGION Network 4: Axis Basics - MC_Home
   #instMcHome(Axis := #axis,   // MC_HOME
               Execute := #homeExecute,
               Position := #homePosition,
               Mode := #homeMode,
               Done => #homeDone,
               Busy => #homeBusy,
               CommandAborted => #statCommandAborted[3],
               Error => #statError[3],
               ErrorId => #statErrorID[3]);
END_REGION

REGION Network 5: Axis Basics - MC_MoveJog
   #instMcMoveJog(Axis := #axis,   // MC_MOVEJOG
                  JogForward := #jogForward,
                  JogBackward := #jogBackward,
                  Velocity := #jogVelocity,
                  Acceleration := #jogAcceleration,
                  Deceleration := #jogDeceleration,
                  Jerk := #jogJerk,
                  PositionControlled := #jogPositionControlled,
                  InVelocity => #jogInVelocity,
                  Busy => #jogBusy,
                  CommandAborted => #statCommandAborted[4],
                  Error => #statError[4],
                  ErrorId => #statErrorID[4]);
END_REGION

REGION Network 6 (SCL): Axis Basics - Generate output signals and error detection
   //General output signals

   //Reset output signals
   #commandAborted := False;
   #error := False;
   #errorID := #ERRORID_DEFAULT;
   #statusID := #STATUSID_DEFAULT;

   //Transfer ARRAY to DWORD
   GATHER(IN:=#statCommandAborted,
          OUT=>#tempDwordCommandAborted);
   GATHER(IN:=#statError,
          OUT=>#tempDwordError);

   //Check for errors or command aborts
   IF (#tempDwordError > DWORD#0)
   THEN
     //Select error information
     FOR #tempCount := #ARRAY_BEGIN TO #ARRAY_END
     DO
       IF (#statError[#tempCount] = True)
       THEN
         #error := True;
         #errorID := #statErrorID[#tempCount];
         #statusID := #tempCount;
         EXIT;
       END_IF;
     END_FOR;
   ELSIF (#tempDwordCommandAborted > DWORD#0)
   THEN
     //Select command aborted information
     FOR #tempCount := #ARRAY_BEGIN TO #ARRAY_END
     DO
       IF (#statCommandAborted[#tempCount] = True)
       THEN
         #commandAborted := True;
         #errorID := #statErrorID[#tempCount];
         #statusID := #tempCount;
         EXIT;
       END_IF;
     END_FOR;
   END_IF;
END_REGION
END_FUNCTION_BLOCK

FUNCTION_BLOCK "SimaHydTO_AxisAdvanced_PosAxis"   // FB33111, FBD
TITLE = SimaHydTO_AxisAdvanced_PosAxis
{ S7_Optimized_Access := 'TRUE' }
FAMILY : SimaHydTO/LAxisBasics
VERSION : 1.0
// Function block information: See Function block network 1
// stored: AutoNumber true, IsIECCheckEnabled false, IsRetainMemResEnabled false, MemoryReserve 100, SetENOAutomatically false, UDAEnableTagReadback false
   VAR_INPUT
      axis : TO_PositioningAxis;   // Technology object (axis)
      moveRelativeExecute : Bool;   // MC_MoveRelative: Start job with a positive edge
      moveRelativeDistance : LReal := 0.0;   // Distance of relative movement
      moveAbsoluteExecute : Bool;   // MC_MoveAbsolute: Start job with a positive edge
      moveAbsolutePosition : LReal := 0.0;   // Target position of absolute movement
      moveAbsoluteDirection : Int := 1;   // Direction of absolute movement: 0: Positive direction / 1: Negative direction / 3: Shortest direction
      moveAbsPositionControlled : Bool := true;   // 0: Non position-controlled operation / 1: Position-controlled mode - The parameter applies as long as the MC_MoveJog command is executed. After this, the setting of MC_Power applies again.
      haltExecute : Bool;   // MC_Halt: Start job with a positive edge
      haltAbortAcceleration : Bool := false;   // Acceleration control: False: The current acceleration at the start of the job is reduced using the configured jerk. Afterwards, the deceleration builds up / True: The acceleration is set to 0.0 at the start of the job, and the deceleration immediately builds up.
      Velocity : LReal := 100.0;   // Velocity of movement
      Acceleration : LReal := -1.0;   // Acceleration of movement
      Deceleration : LReal := -1.0;   // Deceleration of movement
      Jerk : LReal := -1.0;   // Jerk of movement
   END_VAR
   VAR_OUTPUT
      moveRelativeDone { ExternalWritable := 'False'} : Bool;   // MC_MoveRelative: Job is completed
      moveRelativeBusy { ExternalWritable := 'False'} : Bool;   // MC_MoveRelative: Job is running
      moveAbsoluteDone { ExternalWritable := 'False'} : Bool;   // MC_MoveAbsolute: Job is completed
      moveAbsoluteBusy { ExternalWritable := 'False'} : Bool;   // MC_MoveAbsolute: Job is running
      haltDone { ExternalWritable := 'False'} : Bool;   // MC_Halt: Job is running
      haltBusy { ExternalWritable := 'False'} : Bool;   // MC_Halt: Job is running
      commandAborted { ExternalWritable := 'False'} : Bool;   // The job was aborted by another job during execution (see also StatusID)
      error { ExternalWritable := 'False'} : Bool;   // An error occurred during execution of the job. The job is rejected. The cause of the error can be found in the "ErrorID" parameter.
      errorID { ExternalWritable := 'False'} : Word;   // ErrorID of motion control instruction (see also StatusID)
      statusID { ExternalWritable := 'False'} : Int;   // Additional specification of affected Motion control instruction of CommandAborted or Error: 0: No instruction / 1: MC_MoveRelative / 2: MC_MoveAbsolute / 3: MC_Halt
   END_VAR
   VAR
      instMcMoveRelative { ExternalAccessible := 'False'; ExternalVisible := 'False'; ExternalWritable := 'False'; S7_SetPoint := 'True'} : MC_MOVERELATIVE;   // PLCopen functions of basic motion control
      instMcMoveAbsolute { ExternalAccessible := 'False'; ExternalVisible := 'False'; ExternalWritable := 'False'; S7_SetPoint := 'True'} : MC_MOVEABSOLUTE;
      instMcHalt { ExternalAccessible := 'False'; ExternalVisible := 'False'; ExternalWritable := 'False'; S7_SetPoint := 'True'} : MC_HALT;
      statCommandAborted { ExternalAccessible := 'False'; ExternalVisible := 'False'; ExternalWritable := 'False'} : Array[#ARRAY_BEGIN..#ARRAY_END] of Bool;   // Arrays to save error information of PLCopen functions
      statError { ExternalAccessible := 'False'; ExternalVisible := 'False'; ExternalWritable := 'False'} : Array[#ARRAY_BEGIN..#ARRAY_END] of Bool;
      statErrorID { ExternalAccessible := 'False'; ExternalVisible := 'False'; ExternalWritable := 'False'} : Array[#ARRAY_BEGIN..#ARRAY_END] of Word;
      instMoveAbsOpenLoop { S7_SetPoint := 'True'} : "LSimaHydTO_MC_MoveAbsOpenLoop";
   END_VAR
   VAR_TEMP
      tempDwordCommandAborted : DWord;   // Variables to check error informations of PLCopen functions
      tempDwordError : DWord;
      tempCount : Int;   // Counter of FOR counting loop
   END_VAR
   VAR CONSTANT
      ARRAY_BEGIN : Int := 1;   // Start-Index of array (Maximum 32 Array elements!)
      ARRAY_END : Int := 32;   // End-Index of array (Maximum 32 Array elements!)
      ERROR_DEFAULT : Bool := false;   // Default values of output signals
      ERRORID_DEFAULT : Word := 16#0;
      STATUSID_DEFAULT : Int := 0;
   END_VAR
BEGIN

REGION Network 1 (SCL): Axis Basics - Header
   //=============================================================================
   //SIEMENS AG
   //(c)Copyright 2016 All Rights Reserved
   //-----------------------------------------------------------------------------
   //Library:       AxisAdvanced
   //Tested with:   S7-1500 V2.5
   //Engineering:   TIA Portal V15
   //Restrictions:  Motion Control Library V4.0
   //Requirements:  S7-1500(T)
   //Functionality: Advanced axis control of TO_PositioningAxis
   //-----------------------------------------------------------------------------
   //Change log table:
   //Version  Date       Expert in charge Changes applied
   //01.00.00 19.07.2019 ArSc             First released version
   //=============================================================================
END_REGION

REGION Network 2: Axis Advanced - MC_MoveRelative
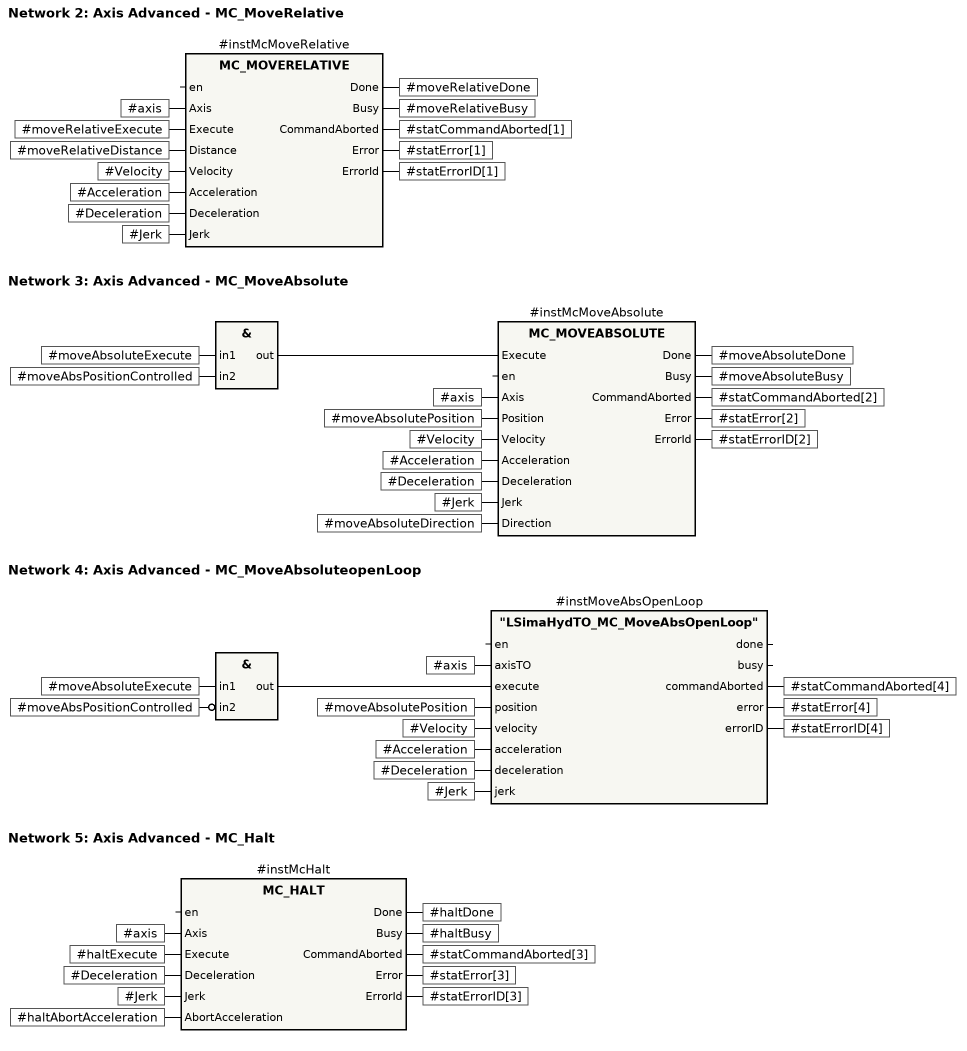
   #instMcMoveRelative(Axis := #axis,   // MC_MOVERELATIVE
                       Execute := #moveRelativeExecute,
                       Distance := #moveRelativeDistance,
                       Velocity := #Velocity,
                       Acceleration := #Acceleration,
                       Deceleration := #Deceleration,
                       Jerk := #Jerk,
                       Done => #moveRelativeDone,
                       Busy => #moveRelativeBusy,
                       CommandAborted => #statCommandAborted[1],
                       Error => #statError[1],
                       ErrorId => #statErrorID[1]);
END_REGION

REGION Network 3: Axis Advanced - MC_MoveAbsolute
   #instMcMoveAbsolute(Execute := #moveAbsoluteExecute AND #moveAbsPositionControlled,   // MC_MOVEABSOLUTE
                       Axis := #axis,
                       Position := #moveAbsolutePosition,
                       Velocity := #Velocity,
                       Acceleration := #Acceleration,
                       Deceleration := #Deceleration,
                       Jerk := #Jerk,
                       Direction := #moveAbsoluteDirection,
                       Done => #moveAbsoluteDone,
                       Busy => #moveAbsoluteBusy,
                       CommandAborted => #statCommandAborted[2],
                       Error => #statError[2],
                       ErrorId => #statErrorID[2]);
END_REGION

REGION Network 4: Axis Advanced - MC_MoveAbsoluteopenLoop
   #instMoveAbsOpenLoop(axisTO := #axis,   // "LSimaHydTO_MC_MoveAbsOpenLoop"
                        execute := #moveAbsoluteExecute AND NOT #moveAbsPositionControlled,
                        position := #moveAbsolutePosition,
                        velocity := #Velocity,
                        acceleration := #Acceleration,
                        deceleration := #Deceleration,
                        jerk := #Jerk,
                        commandAborted => #statCommandAborted[4],
                        error => #statError[4],
                        errorID => #statErrorID[4]);
END_REGION

REGION Network 5: Axis Advanced - MC_Halt
   #instMcHalt(Axis := #axis,   // MC_HALT
               Execute := #haltExecute,
               Deceleration := #Deceleration,
               Jerk := #Jerk,
               AbortAcceleration := #haltAbortAcceleration,
               Done => #haltDone,
               Busy => #haltBusy,
               CommandAborted => #statCommandAborted[3],
               Error => #statError[3],
               ErrorId => #statErrorID[3]);
END_REGION

REGION Network 6 (SCL): Axis Basics - Generate output signals and error detection
   //General output signals

   //Reset output signals
   #commandAborted := False;
   #error := False;
   #errorID := #ERRORID_DEFAULT;
   #statusID := #STATUSID_DEFAULT;

   //Transfer ARRAY to DWORD
   GATHER(IN:=#statCommandAborted,
          OUT=>#tempDwordCommandAborted);
   GATHER(IN:=#statError,
          OUT=>#tempDwordError);

   //Check for errors or command aborts
   IF (#tempDwordError > DWORD#0)
   THEN
     //Select error information
     FOR #tempCount := #ARRAY_BEGIN TO #ARRAY_END
     DO
       IF (#statError[#tempCount] = True)
       THEN
         #error := True;
         #errorID := #statErrorID[#tempCount];
         #statusID := #tempCount;
         EXIT;
       END_IF;
     END_FOR;
   ELSIF (#tempDwordCommandAborted > DWORD#0)
   THEN
     //Select command aborted information
     FOR #tempCount := #ARRAY_BEGIN TO #ARRAY_END
     DO
       IF (#statCommandAborted[#tempCount] = True)
       THEN
         #commandAborted := True;
         #errorID := #statErrorID[#tempCount];
         #statusID := #tempCount;
         EXIT;
       END_IF;
     END_FOR;
   END_IF;
END_REGION
END_FUNCTION_BLOCK

FUNCTION_BLOCK "LSimaHydTO_MC_MoveAbsOpenLoop"
{ S7_Optimized_Access := 'TRUE' }
AUTHOR : APC_ERLF
FAMILY : LSimaHydTO
VERSION : 1.22
   VAR_INPUT 
      axisTO {InstructionName := 'TO_PositioningAxis'; LibVersion := '4.0'} : TO_PositioningAxis;
      execute : Bool;
      position : LReal;
      velocity : LReal := 100.0;
      acceleration : LReal := 100.0;
      deceleration : LReal := 100.0;
      jerk : LReal := 100.0;
   END_VAR

   VAR_OUTPUT 
      done { ExternalWritable := 'False'} : Bool;
      busy { ExternalWritable := 'False'} : Bool;
      commandAborted { ExternalWritable := 'False'} : Bool;
      error { ExternalWritable := 'False'} : Bool;
      errorID { ExternalWritable := 'False'} : Word;
   END_VAR

   VAR 
      statFBState { ExternalAccessible := 'False'; ExternalVisible := 'False'; ExternalWritable := 'False'} : DInt;
      statExecuteOld { ExternalAccessible := 'False'; ExternalVisible := 'False'; ExternalWritable := 'False'} : Bool;
      instMcMoveVelocity {InstructionName := 'MC_MOVEVELOCITY'; LibVersion := '4.0'; ExternalAccessible := 'False'; ExternalVisible := 'False'; ExternalWritable := 'False'} : MC_MOVEVELOCITY;
      statPosition { ExternalAccessible := 'False'; ExternalVisible := 'False'; ExternalWritable := 'False'} : LReal;
      statVelocity { ExternalAccessible := 'False'; ExternalVisible := 'False'; ExternalWritable := 'False'} : LReal;
      statAcceleration { ExternalAccessible := 'False'; ExternalVisible := 'False'; ExternalWritable := 'False'} : LReal;
      statDeceleration { ExternalAccessible := 'False'; ExternalVisible := 'False'; ExternalWritable := 'False'} : LReal;
      statDecelNorm { ExternalAccessible := 'False'; ExternalVisible := 'False'; ExternalWritable := 'False'} : LReal;
      statJerk { ExternalAccessible := 'False'; ExternalVisible := 'False'; ExternalWritable := 'False'} : LReal;
      statDirection { ExternalAccessible := 'False'; ExternalVisible := 'False'; ExternalWritable := 'False'} : Int;
      statPosWindow { ExternalAccessible := 'False'; ExternalVisible := 'False'; ExternalWritable := 'False'} : LReal;
      statActualPosition { ExternalAccessible := 'False'; ExternalVisible := 'False'; ExternalWritable := 'False'} : LReal;
      statActualVelNorm { ExternalAccessible := 'False'; ExternalVisible := 'False'; ExternalWritable := 'False'} : LReal;
      statStopDistance { ExternalAccessible := 'False'; ExternalVisible := 'False'; ExternalWritable := 'False'} : LReal;
      instTON_Deceleration {InstructionName := 'TON_TIME'; LibVersion := '1.0'; ExternalAccessible := 'False'; ExternalVisible := 'False'; ExternalWritable := 'False'} : TON_TIME;
      statTimeDelay { ExternalAccessible := 'False'; ExternalVisible := 'False'; ExternalWritable := 'False'} : Time;
      statElapsedDelayTime { ExternalAccessible := 'False'; ExternalVisible := 'False'; ExternalWritable := 'False'} : LReal;
      statDecelOpenLoop { ExternalAccessible := 'False'; ExternalVisible := 'False'; ExternalWritable := 'False'} : LReal;
      statMaxDeceleration { ExternalAccessible := 'False'; ExternalVisible := 'False'; ExternalWritable := 'False'} : LReal;
      statLengthUnit { ExternalAccessible := 'False'; ExternalVisible := 'False'; ExternalWritable := 'False'} : UDInt;
      statVelocityUnit { ExternalAccessible := 'False'; ExternalVisible := 'False'; ExternalWritable := 'False'} : UDInt;
      statIntVelocityFactor { ExternalAccessible := 'False'; ExternalVisible := 'False'; ExternalWritable := 'False'} : LReal := 1.0;
      statIntAccFactor { ExternalAccessible := 'False'; ExternalVisible := 'False'; ExternalWritable := 'False'} : LReal := 1.0;
   END_VAR

   VAR CONSTANT 
      NO_ERROR : Word := 16#0000_0000;
      STATE_IDLE : DInt;
      STATE_FIRST_CYCLE : DInt := 10;
      STATE_BUSY : DInt := 20;
      STATE_DECELERATION : DInt := 23;
      STATE_FINISHING : DInt := 25;
      STATE_DONE : DInt := 30;
      STATE_COMMAND_ABORTED : DInt := 40;
      STATE_ERROR : DInt := 100;
   END_VAR


BEGIN
	//================================================================================
	//SIEMENS AG // (c)Copyright 2019 All Rights Reserved
	//--------------------------------------------------------------------------------
	//Library:       LSimaHydTO
	//Tested with:   S7-15xx
	//Engineering:   TIA Portal  V15
	//Restrictions:  -
	//Requirements:  S7-1500 (FW 2.5)
	//Functionality: Function starts the positioning motion of an axis to
	//               an absolute position with open loop position controller.
	//
	//--------------------------------------------------------------------------------
	//Change log table:
	//
	//Version     Date          Expert in charge    Changes applied
	//01.00.00    15.03.2018    APC_ERLF            First released version
	//01.22    22.04.2020    APC_ERLF              - improved: units are taken into account for the control
	
	//================================================================================
	
	
	//----------------------------------------------------------------------
	//start
	//----------------------------------------------------------------------
	
	// rising edge of execute starts functionality
	IF #execute AND NOT #statExecuteOld THEN
	  // initialization
	  #done := FALSE;
	  #commandAborted := FALSE;
	  #busy := FALSE;
	  #error := FALSE;
	  #errorID := #NO_ERROR;
	  IF #axisTO.PositionLimits_SW.Active THEN
	    IF #position > #axisTO.PositionLimits_SW.MaxPosition THEN
	      #statPosition := #axisTO.PositionLimits_SW.MaxPosition;
	    ELSIF #position < #axisTO.PositionLimits_SW.MinPosition THEN
	      #statPosition := #axisTO.PositionLimits_SW.MinPosition;
	    ELSE
	      #statPosition := #position;
	    END_IF;
	  ELSE
	    #statPosition := #position;
	  END_IF;
	  
	  #statLengthUnit := #axisTO.Units.LengthUnit;
	  #statVelocityUnit := #axisTO.Units.VelocityUnit;
	  
	  #statIntVelocityFactor := "LSimaHydTO_GetUnitsCorrection"(lengthUnit := #statLengthUnit,
	                                                            velocityUnit := #statVelocityUnit,
	                                                            accelFactor => #statIntAccFactor);
	  
	  IF #velocity < 0.0 THEN
	      #statVelocity := #axisTO.DynamicDefaults.Velocity;
	  ELSE
	      #statVelocity := ABS(#velocity);
	  END_IF;
	  #statAcceleration := #acceleration;
	  IF #deceleration < 0.0 THEN
	    #statDeceleration := #axisTO.DynamicDefaults.Deceleration;
	  ELSE
	    #statDeceleration := #deceleration;
	  END_IF;
	  #statDecelNorm := #statDeceleration / #statIntAccFactor;
	  #statJerk := #jerk;
	  IF #statPosition > #axisTO.ActualPosition THEN
	    #statDirection := 1; // positive
	  ELSIF #statPosition < #axisTO.ActualPosition THEN
	    #statDirection := 2; // negative
	  END_IF;
	  
	  #statPosWindow := #axisTO.PositioningMonitoring.Window;
	  #statMaxDeceleration := #axisTO.DynamicLimits.MaxDeceleration * 0.999;
	  #instMcMoveVelocity(Axis := #axisTO,
	                            Execute := FALSE,
	                            Velocity := #statVelocity,
	                            Acceleration := #statAcceleration,
	                            Deceleration := #statDeceleration,
	                            Jerk := #statJerk,
	                            Direction := #statDirection,
	                            Current := FALSE,
	                            PositionControlled := FALSE);
	  
	  #statFBState := #STATE_BUSY;
	END_IF;
	
	
	//----------------------------------------------------------------------
	//busy
	//----------------------------------------------------------------------
	// state machine
	// ------------------------------------------------------------------
	CASE #statFBState OF
	    
	    
	  #STATE_FIRST_CYCLE:
	    
	    ;
	    
	    
	  #STATE_BUSY:
	    
	    
	    #instMcMoveVelocity(Axis := #axisTO,
	                              Execute := TRUE,
	                              Velocity := #statVelocity,
	                              Acceleration := #statAcceleration,
	                              Deceleration := #statDeceleration,
	                              Jerk := #statJerk,
	                              Direction := #statDirection,
	                              Current := FALSE,
	                              PositionControlled := FALSE,
	                              Busy => #busy,
	                              CommandAborted => #commandAborted,
	                              Error => #error,
	                              ErrorId => #errorID);
	    
	    IF #error THEN
	      #statFBState := #STATE_ERROR;
	    ELSIF #busy THEN
	      #statActualPosition := #axisTO.ActualPosition;
	      #statActualVelNorm := ABS(#axisTO.ActualVelocity)/#statIntVelocityFactor;
	      #statStopDistance := #axisTO.DynamicAxisModel.VelocityTimeConstant * #statActualVelNorm +
	                          (#statActualVelNorm * ABS(#axisTO.Velocity)/#statIntVelocityFactor) / (2.0 * #statDecelNorm);
	      IF (#statDirection = 1 AND #statActualPosition >= (#statPosition - #statPosWindow))
	        OR (#statDirection = 2 AND #statActualPosition <= (#statPosition + #statPosWindow)) THEN
	        
	        #instMcMoveVelocity(Axis := #axisTO,
	                                  Execute := FALSE);
	        
	        #statFBState := #STATE_FINISHING;
	      ELSIF (#statDirection = 1 AND #statActualPosition >= (#statPosition - #statStopDistance))
	        OR (#statDirection = 2 AND #statActualPosition <= (#statPosition + #statStopDistance))
	       THEN 
	        
	        #instMcMoveVelocity(Axis := #axisTO,
	                                  Execute := FALSE);
	        
	        #statTimeDelay := LREAL_TO_DINT(#axisTO.DynamicAxisModel.VelocityTimeConstant * 1000.0);
	        #statVelocity := SQRT(2.0 * #axisTO.PositioningMonitoring.Window * #statDecelNorm)*#statIntVelocityFactor;
	        
	        #instTON_Deceleration(IN := FALSE,
	                          PT := #statTimeDelay);
	        
	        #statFBState := #STATE_DECELERATION;
	      END_IF;
	    ELSIF #commandAborted THEN
	      #statFBState := #STATE_COMMAND_ABORTED;
	    END_IF;
	    
	    
	  #STATE_DECELERATION:
	    
	    #instMcMoveVelocity(Axis := #axisTO,
	                              Execute := FALSE,
	                              Busy => #busy,
	                              CommandAborted => #commandAborted,
	                              Error => #error,
	                              ErrorId => #errorID);
	    
	    IF #error THEN
	      #statFBState := #STATE_ERROR;
	    ELSIF #busy THEN
	      #statActualPosition := #axisTO.ActualPosition;
	      #statActualVelNorm := ABS(#axisTO.ActualVelocity)/#statIntVelocityFactor;
	      
	      IF (#statDirection = 1 AND #statActualPosition >= (#statPosition - #statPosWindow))
	        OR (#statDirection = 2 AND #statActualPosition <= (#statPosition + #statPosWindow)) THEN
	        
	        #instMcMoveVelocity(Axis := #axisTO,
	                                  Execute := FALSE);
	        
	        #statFBState := #STATE_FINISHING;
	      ELSE
	        
	        #instTON_Deceleration(IN := TRUE,
	                          PT := #statTimeDelay);
	        
	        #statElapsedDelayTime := LIMIT(MN := 0.0,
	                                       IN := TIME_TO_DINT(#statTimeDelay - #instTON_Deceleration.ET),
	                                       MX := TIME_TO_DINT(#statTimeDelay))*0.001;
	        #statDecelOpenLoop := LIMIT(MN:= 0.1*#statDeceleration,
	                                    IN := #statIntAccFactor *(#statActualVelNorm * ABS(#axisTO.Velocity)/#statIntVelocityFactor) /
	                                        (2.0 * (ABS(#statActualPosition - #statPosition) - #statElapsedDelayTime * #statActualVelNorm)),
	                                    MX := #statMaxDeceleration);
	        
	        #instMcMoveVelocity(Axis := #axisTO,
	                                  Execute := TRUE,
	                                  Velocity := #statVelocity,
	                                  Acceleration := #statAcceleration,
	                                  Deceleration := #statDecelOpenLoop,
	                                  Jerk := 0.0,
	                                  Direction := #statDirection,
	                                  Current := FALSE,
	                                  PositionControlled := FALSE,
	                                  Busy => #busy,
	                                  CommandAborted => #commandAborted,
	                                  Error => #error,
	                                  ErrorId => #errorID);
	        
	        IF #error THEN
	          #statFBState := #STATE_ERROR;
	        END_IF;
	      END_IF;
	    ELSIF #commandAborted THEN
	      #statFBState := #STATE_COMMAND_ABORTED;
	    END_IF;
	    
	    
	  #STATE_FINISHING:
	    
	    #instMcMoveVelocity(Axis := #axisTO,
	                              Execute := TRUE,
	                              Velocity := 0.0,
	                              Acceleration := #statAcceleration,
	                              Deceleration := #statDeceleration,
	                              Jerk := 0.0,
	                              Direction := 0, //statDirection,
	                              Current := FALSE,
	                              PositionControlled := FALSE,
	                              Busy => #busy,
	                              CommandAborted => #commandAborted,
	                              Error => #error,
	                              ErrorId => #errorID);
	    
	    IF #error THEN
	      #statFBState := #STATE_ERROR;
	    ELSIF #commandAborted THEN
	      #statFBState := #STATE_COMMAND_ABORTED;
	    ELSIF NOT #busy OR #instMcMoveVelocity.InVelocity THEN
	      #busy := FALSE;
	      #done := TRUE;
	      #statFBState := #STATE_DONE;
	    END_IF;
	    
	
	  #STATE_IDLE:
	    
	    //==================================================================
	    //state analysis (no function)
	    //==================================================================
	    
	    ;
	    
	    
	  #STATE_DONE:
	    
	    //==================================================================
	    //output for one cycle minimum
	    //==================================================================
	    
	    IF NOT #execute THEN
	      #done := FALSE;
	      #statFBState := #STATE_IDLE;
	    END_IF;
	    
	    
	  #STATE_COMMAND_ABORTED:
	    
	    //==================================================================
	    //reset commandAborted, output for one cycle minimum
	    //==================================================================
	    
	    IF NOT #execute THEN
	      #commandAborted := FALSE;
	      #statFBState := #STATE_IDLE;
	    END_IF;
	    
	    
	  #STATE_ERROR:
	    //==================================================================
	    //reset error, output for one cycle minimum
	    //==================================================================
	    
	    IF NOT #execute THEN
	      #error := FALSE;
	      #errorID := #NO_ERROR;
	      #statFBState := #STATE_IDLE;
	    END_IF;
	    
	    
	  ELSE
	    //==================================================================
	    //when FB is busy...
	    //==================================================================
	    
	    ;
	    
	END_CASE;
	
	//-------------------------------------------------------------------------
	//always executed
	//-------------------------------------------------------------------------
	
	// edge detection
	#statExecuteOld := #execute;
	// ------------------------------------------------------------------------------
END_FUNCTION_BLOCK

FUNCTION_BLOCK "LSimaHydTO_HydraulicSimulationAnalog"
{ S7_Optimized_Access := 'TRUE' }
AUTHOR : APC_ERLF
FAMILY : LSimaHydTO
VERSION : 1.22
   VAR_INPUT 
      enable : Bool;
      analogInput : Int;
      initPosition : LReal;
      minPosition : LReal := -1000000000000.0;
      maxPosition : LReal := 1000000000000.0;
      maxVelocity : LReal := 500.0;
      maxForce : LReal := 100.0;
      springDistance : LReal := 1.0;
      externalForce : LReal := 0.0;
      dynamicFrictionFactor : LReal;
      fixedStop : LReal := 1000000000000.0;
      fixedStopInverse : Bool;
      forceInverse : Bool;
      delayTime : LReal;
      cycleTime : UDInt;
      vChar_DB_NUMBER : UInt;
      axisTO : DB_ANY;
      Pozisyon_Input : LReal;
   END_VAR

   VAR_OUTPUT 
      busy { ExternalWritable := 'False'} : Bool;
      active { ExternalWritable := 'False'} : Bool;
      error { ExternalWritable := 'False'} : Bool;
      status { ExternalWritable := 'False'} : Word;
      simulatedPosition { ExternalWritable := 'False'} : LReal;
      simulatedForce { ExternalWritable := 'False'} : LReal;
      simulatedVChar { ExternalWritable := 'False'} : UInt;
      forceSensorAnalog_A { ExternalWritable := 'False'} : Word;
      forceSensorAnalog_B { ExternalWritable := 'False'} : Word;
   END_VAR

   VAR_IN_OUT 
      tel81in {InstructionName := 'PD_TEL81_IN'; LibVersion := '4.0'} : PD_TEL81_IN;
      tel81out {InstructionName := 'PD_TEL81_OUT'; LibVersion := '4.0'} : PD_TEL81_OUT;
   END_VAR

   VAR 
      statSetPoint { ExternalAccessible := 'False'; ExternalVisible := 'False'; ExternalWritable := 'False'} : LReal;
      statVelSetPoint { ExternalAccessible := 'False'; ExternalVisible := 'False'; ExternalWritable := 'False'} : LReal;
      statActualVChar { ExternalAccessible := 'False'; ExternalVisible := 'False'; ExternalWritable := 'False'} : UInt;
      statSampleTime { ExternalAccessible := 'False'; ExternalVisible := 'False'; ExternalWritable := 'False'} : LReal;
      statActualPosition { ExternalAccessible := 'False'; ExternalVisible := 'False'; ExternalWritable := 'False'} : LReal;
      statActualForce { ExternalAccessible := 'False'; ExternalVisible := 'False'; ExternalWritable := 'False'} : LReal;
      statForceFactor { ExternalAccessible := 'False'; ExternalVisible := 'False'; ExternalWritable := 'False'} : LReal;
      statEnableOld { ExternalAccessible := 'False'; ExternalVisible := 'False'; ExternalWritable := 'False'} : Bool;
      instSetPointPT1 { ExternalAccessible := 'False'; ExternalVisible := 'False'; ExternalWritable := 'False'} : "LSimaHydTO_T1";
      statPosLimitForce { ExternalAccessible := 'False'; ExternalVisible := 'False'; ExternalWritable := 'False'} : LReal;
      statNegLimitForce { ExternalAccessible := 'False'; ExternalVisible := 'False'; ExternalWritable := 'False'} : LReal;
      statFrictionForce { ExternalAccessible := 'False'; ExternalVisible := 'False'; ExternalWritable := 'False'} : LReal;
      instSimpleEncSetValue { ExternalAccessible := 'False'; ExternalVisible := 'False'; ExternalWritable := 'False'} : "LSimaHydTO_SimpleEncTel81";
      statVCharDB { ExternalAccessible := 'False'; ExternalVisible := 'False'; ExternalWritable := 'False'} : DB_ANY;
      statErrorVariant { ExternalAccessible := 'False'; ExternalVisible := 'False'; ExternalWritable := 'False'} : Int;
      statIntVelocityFactor { ExternalAccessible := 'False'; ExternalVisible := 'False'; ExternalWritable := 'False'} : LReal := 1.0;
   END_VAR

   VAR_TEMP 
      tempDeltaPosition : LReal;
      tempMinPos : LReal;
      tempMaxPos : LReal;
      tempActPosOld : LReal;
      tempVCharVar : Variant;
      tempRefToVChar : REF_TO "LSimaHydTO_typeVCharData";
      tempAccFactor : LReal;
   END_VAR

   VAR CONSTANT 
      ERR_INVALID_TYPE_OF_AXIS : Word := 16#8201;
   END_VAR


BEGIN
	//================================================================================
	//SIEMENS AG // (c)Copyright 2019 All Rights Reserved
	//--------------------------------------------------------------------------------
	//Library:       LSimaHydTO
	//Tested with:   S7-15xx
	//Engineering:   TIA Portal  V15
	//Restrictions:  -
	//Requirements:  S7-1500 (FW 2.5)
	//Functionality: Simulation of hydraulic cylinder   
	//
	//--------------------------------------------------------------------------------
	//Change log table:
	//
	//Version     Date          Expert in charge    Changes applied
	//01.00    15.03.2018    APC_ERLF            First released version
	//01.22    22.04.2020    APC_ERLF            improved: units are taken into account for the control
	//================================================================================
	
	
	IF #enable THEN
	    IF NOT #statEnableOld THEN //positive edge at enable
	        #error := FALSE;
	        #status := 16#0000;
	        #statSampleTime := UDINT_TO_LREAL(#cycleTime) * lreal#1.0E-9;
	       #statActualPosition := #initPosition;
	        
	        CASE TypeOfDB(#axisTO) OF
	                
	            TO_PositioningAxis:
	                #statIntVelocityFactor := "LSimaHydTO_GetPosAxisCorrection"(axis := #axisTO, accelFactor => #tempAccFactor);
	                
	            TO_SynchronousAxis:
	                #statIntVelocityFactor := "LSimaHydTO_GetSyncAxisCorrection"(axis := #axisTO, accelFactor => #tempAccFactor);
	                
	            ELSE
	                #error := TRUE;
	                #status := #ERR_INVALID_TYPE_OF_AXIS; // erorr
	                RETURN;
	        END_CASE;
	        
	        #busy := TRUE;
	        #active := TRUE;
	        
	        
	    END_IF;
	    REGION evaluteVChar
	        IF #vChar_DB_NUMBER > 0 THEN
	            #statVCharDB := UINT_TO_DB_ANY(#vChar_DB_NUMBER);
	            #tempVCharVar := DB_ANY_TO_VARIANT(in := #statVCharDB, err => #statErrorVariant);
	            IF #statErrorVariant = 0 THEN
	                #tempRefToVChar ?= #tempVCharVar;
	                
	                IF TypeOf(#tempVCharVar) <> LSimaHydTO_typeVCharData THEN
	                    #statErrorVariant := 8200;
	                END_IF;
	            END_IF;
	            IF #statErrorVariant <> 0 THEN
	                #statActualVChar := 0;
	                
	            ELSE
	                // check consinsesty of VChar
	                IF #tempRefToVChar^.MaxIdx < 1 OR #tempRefToVChar^.VelocityLimitPositive <= #tempRefToVChar^.VelocityLimitNegative THEN
	                    #statActualVChar := 0;
	                ELSE
	                    #statActualVChar := #vChar_DB_NUMBER;
	                END_IF;
	            END_IF;
	        ELSE
	            #statActualVChar := 0;
	        END_IF;
	        
	        
	        
	        #statSetPoint := lreal#0.0036168981 * INT_TO_LREAL(#analogInput);
	        
	        IF #statActualVChar = 0 THEN
	            #statVelSetPoint := "LSimaHydTO_Scale"(input := #statSetPoint,
	                                                   inBegin := -100.0,
	                                                   inEnd := 100.0,
	                                                   valBegin := - #maxVelocity,
	                                                   valEnd := #maxVelocity);
	        ELSE
	            
	            #statVelSetPoint := "LSimaHydTO_VcharInverse"(qOutput := #statSetPoint, VChar := #tempRefToVChar^);
	            
	            #statVelSetPoint := LIMIT(MN := - #maxVelocity, IN := #statVelSetPoint, MX := #maxVelocity);
	        END_IF;
	        #statVelSetPoint := #statVelSetPoint / #statIntVelocityFactor;
	        #simulatedVChar := #statActualVChar;
	    END_REGION
	    
	    #statActualForce := LIMIT(MN := - #maxForce, IN := #statActualForce, MX := #maxForce);
	    IF (#statActualForce > 0.0 AND
	        #statVelSetPoint > 0.0)
	        OR
	        (#statActualForce < 0.0 AND
	        #statVelSetPoint < 0.0)
	    THEN
	        #statForceFactor := MAX(IN1 := 0.0, IN2 := SQRT((#maxForce - ABS(#statActualForce)) / #maxForce));
	    ELSE
	        #statForceFactor := 1.0;
	    END_IF;
	    
	    
	    #instSetPointPT1(enable := #enable AND #delayTime > 0.0,
	                     inputValue := #statVelSetPoint,
	                     timeConstant := #delayTime,
	                     sampleTime := #statSampleTime
	                     // ,outputValue => 
	                     // ,active => 
	                     // ,error => 
	    );
	    
	    #tempDeltaPosition := (#instSetPointPT1.outputValue) * #statSampleTime * #statForceFactor;
	    
	    //calculate AND LIMIT actual postition
	    #tempActPosOld := #statActualPosition;
	    
	    IF #fixedStopInverse THEN
	        #tempMinPos := LIMIT(MN := #minPosition
	                             , IN := #fixedStop
	                             , MX := #maxPosition);
	        #tempMaxPos := #maxPosition;
	    ELSE
	        #tempMinPos := #minPosition;
	        #tempMaxPos := LIMIT(MN := #minPosition
	                             , IN := #fixedStop
	                             , MX := #maxPosition);
	        
	    END_IF;
	    (*#statActualPosition := LIMIT(MN := #tempMinPos
	                                 , IN := #tempActPosOld + #tempDeltaPosition
	                                 , MX := #tempMaxPos
	    );*)
	    #statActualPosition := #Pozisyon_Input;
	    
	    #statFrictionForce := #dynamicFrictionFactor * (#statActualPosition - #tempActPosOld) / #statSampleTime;
	    IF #maxForce > 0.0
	        AND #springDistance > 0.0
	    THEN
	        
	        IF (#tempMaxPos - #statActualPosition) < #springDistance THEN
	            
	            #statPosLimitForce := LIMIT(MN := 0.0
	                                        , IN := (1 - (#tempMaxPos - #statActualPosition) / #springDistance) * #maxForce
	                                        , MX := #maxForce);
	        ELSE
	            #statPosLimitForce := 0.0;
	        END_IF;
	        IF (#statActualPosition - #tempMinPos) < #springDistance THEN
	            #statNegLimitForce := - LIMIT(MN := 0.0
	                                          , IN := (1 - (#statActualPosition - #tempMinPos) / #springDistance) * #maxForce
	                                          , MX := #maxForce);
	        ELSE
	            #statNegLimitForce := 0.0;
	        END_IF;
	        
	        #statActualForce := #externalForce + #statNegLimitForce + #statPosLimitForce + #statFrictionForce;
	        
	    ELSE
	        #statActualForce := #externalForce + #statFrictionForce;
	    END_IF;
	    
	    IF #forceInverse THEN
	        #statActualForce := -1.0 * #statActualForce;
	    END_IF;
	    //write actual position to technology object
	    
	    #simulatedPosition := #statActualPosition;
	    //#simulatedPosition := #Pozisyon_Input;
	    #simulatedForce := LIMIT(MN := - #maxForce, IN := #statActualForce, MX := #maxForce);
	    
	    IF #maxForce > 0.0 THEN
	        IF #simulatedForce >= 0.0 THEN
	            #forceSensorAnalog_A := INT_TO_WORD(LREAL_TO_INT(#simulatedForce * 27648.0 / #maxForce));
	            #forceSensorAnalog_B := 0;
	        ELSE
	            #forceSensorAnalog_B := INT_TO_WORD(LREAL_TO_INT(ABS(#simulatedForce) * 27648.0 / #maxForce));
	            #forceSensorAnalog_A := 0;
	        END_IF;
	    ELSE
	        #forceSensorAnalog_A := 0;
	        #forceSensorAnalog_B := 0;
	    END_IF;
	    
	    #instSimpleEncSetValue(position := #simulatedPosition,
	                           init := #enable AND NOT #statEnableOld,
	                           axis := #axisTO,
	                           status => #status,
	                           tel81in := #tel81in,
	                           tel81out := #tel81out);
	    
	    
	    
	ELSE
	    IF #statEnableOld THEN //negative edge
	        #busy := FALSE;
	        #active := FALSE;
	        #simulatedVChar := 0;
	        
	        #statActualPosition := 0.0;
	        #statActualForce := 0.0;
	        #simulatedPosition := 0.0;
	        #simulatedForce := 0.0;
	        #forceSensorAnalog_A := 0;
	        #forceSensorAnalog_B := 0;
	        
	    END_IF;
	END_IF;
	
	
	#statEnableOld := #enable;
	
	
	
	
	
	
END_FUNCTION_BLOCK

FUNCTION_BLOCK "LSimaHydTO_SimpleEncTel81"
{ S7_Optimized_Access := 'TRUE' }
AUTHOR : APC_ERLF
FAMILY : LSimaHydTO
VERSION : 1.0
   VAR_INPUT 
      init { ExternalAccessible := 'False'; ExternalVisible := 'False'; ExternalWritable := 'False'} : Bool;
      position { ExternalAccessible := 'False'; ExternalVisible := 'False'; ExternalWritable := 'False'} : LReal;
      axis { ExternalAccessible := 'False'; ExternalVisible := 'False'; ExternalWritable := 'False'} : DB_ANY;
   END_VAR

   VAR_OUTPUT 
      status { ExternalAccessible := 'False'; ExternalVisible := 'False'; ExternalWritable := 'False'} : Word;
   END_VAR

   VAR_IN_OUT 
      tel81in {InstructionName := 'PD_TEL81_IN'; LibVersion := '4.0'} : PD_TEL81_IN;
      tel81out {InstructionName := 'PD_TEL81_OUT'; LibVersion := '4.0'} : PD_TEL81_OUT;
   END_VAR

   VAR 
      statInitDone { ExternalAccessible := 'False'; ExternalVisible := 'False'; ExternalWritable := 'False'} : Bool;
      statInitOld { ExternalAccessible := 'False'; ExternalVisible := 'False'; ExternalWritable := 'False'} : Bool;
      statInverseDirection { ExternalAccessible := 'False'; ExternalVisible := 'False'; ExternalWritable := 'False'} : Bool;
      statSensorSystem { ExternalAccessible := 'False'; ExternalVisible := 'False'; ExternalWritable := 'False'} : DInt;
      statMotionType { ExternalAccessible := 'False'; ExternalVisible := 'False'; ExternalWritable := 'False'} : DInt;
      statLeadScrew { ExternalAccessible := 'False'; ExternalVisible := 'False'; ExternalWritable := 'False'} : LReal := 1.0;
      statModulo {InstructionName := 'TO_Struct_Modulo'; LibVersion := '4.0'; ExternalAccessible := 'False'; ExternalVisible := 'False'; ExternalWritable := 'False'} : TO_Struct_Modulo := ((), (), 360.0);
      statSensorParameter {InstructionName := 'TO_Struct_SensorParameter'; LibVersion := '4.0'; ExternalAccessible := 'False'; ExternalVisible := 'False'; ExternalWritable := 'False'} : TO_Struct_SensorParameter;
      statError { ExternalAccessible := 'False'; ExternalVisible := 'False'; ExternalWritable := 'False'} : Bool := FALSE;
      statOldPos { ExternalAccessible := 'False'; ExternalVisible := 'False'; ExternalWritable := 'False'} : LReal;
      statResolutionAbs { ExternalAccessible := 'False'; ExternalVisible := 'False'; ExternalWritable := 'False'} : LReal;
      statResolutionCycl { ExternalAccessible := 'False'; ExternalVisible := 'False'; ExternalWritable := 'False'} : LReal;
      statDIncPos { ExternalAccessible := 'False'; ExternalVisible := 'False'; ExternalWritable := 'False'} : LReal;
      statIncPos { ExternalAccessible := 'False'; ExternalVisible := 'False'; ExternalWritable := 'False'} : DInt;
   END_VAR

   VAR_TEMP 
      tempReqCmd : Bool;
      tempDPos : LReal;
      tempIncResolution : UDInt;
      tempDIncPosInt : DInt;
   END_VAR

   VAR CONSTANT 
      DWORD_1 : DWord := 16#0000_0001;
      ERR_INVALID_TYPE_OF_AXIS : Word := 16#8201;
   END_VAR


BEGIN
	//================================================================================
	//SIEMENS AG // (c)Copyright 2019 All Rights Reserved
	//--------------------------------------------------------------------------------
	//Library:       LSimaHydTO
	// Tested with:     S7-1500 FW V2.0 or higher
	// Engineering:     TIA Portal V14
	// Restrictions:    -
	// Functionality:   set value of the encoder telegramm 81 
	//-----------------------------------------------------------------------------
	// Change log table:
	// Version    Date          Changes applied
	// 01.00.00   12.01.2018    First released version
	//=============================================================================
	
	IF NOT #statInitDone OR (#init AND NOT #statInitOld) THEN
	    #statError := FALSE;
	    #status := 0;
	    CASE TypeOfDB(#axis) OF
	            
	        TO_ExternalEncoder:
	            "LSimaHydTO_GetExternalEncoderData"(axis := #axis,
	                                                inverseDirection => #statInverseDirection,
	                                                sensorSystem => #statSensorSystem,
	                                                motionType => #statMotionType,
	                                                leadScrew => #statLeadScrew,
	                                                modulo => #statModulo,
	                                                sensorParameter => #statSensorParameter);
	            
	            
	        TO_PositioningAxis:
	            #status := "LSimaHydTO_GetPosAxisEncoderData"(axis := #axis,
	                                                          inverseDirection => #statInverseDirection,
	                                                          sensorSystem => #statSensorSystem,
	                                                          motionType => #statMotionType,
	                                                          leadScrew => #statLeadScrew,
	                                                          modulo => #statModulo,
	                                                          sensorParameter => #statSensorParameter);
	            
	        TO_SynchronousAxis:
	            #status := "LSimaHydTO_GetSyncAxisEncoderData"(axis := #axis,
	                                                           inverseDirection => #statInverseDirection,
	                                                           sensorSystem => #statSensorSystem,
	                                                           motionType => #statMotionType,
	                                                           leadScrew => #statLeadScrew,
	                                                           modulo => #statModulo,
	                                                           sensorParameter => #statSensorParameter);
	            
	        ELSE
	            #status := #ERR_INVALID_TYPE_OF_AXIS; // erorr
	    END_CASE;
	    
	    IF #status = 0 THEN
	        
	        IF #statSensorSystem = 0 THEN
	            //linear encoder
	            #tempIncResolution := DWORD_TO_UDINT(SHL(IN := #DWORD_1, N := #statSensorParameter.FineResolutionXist1));
	            #statResolutionCycl := #tempIncResolution / #statSensorParameter.Resolution;
	            #tempIncResolution := DWORD_TO_UDINT(SHL(IN := #DWORD_1, N := #statSensorParameter.FineResolutionXist2));
	            #statResolutionAbs := #tempIncResolution / #statSensorParameter.Resolution;
	            
	        ELSIF #statSensorSystem = 1 THEN
	            //rotatory encoder
	            #tempIncResolution := #statSensorParameter.StepsPerRevolution * DWORD_TO_UDINT(SHL(IN := #DWORD_1, N := #statSensorParameter.FineResolutionXist1));
	            IF #statMotionType = 0 THEN
	                //linear axis
	                #statResolutionCycl := #tempIncResolution / #statLeadScrew;
	            ELSE
	                // rotatory axis
	                #statResolutionCycl := #tempIncResolution / 360.0;
	            END_IF;
	            #tempIncResolution := #statSensorParameter.StepsPerRevolution * DWORD_TO_UDINT(SHL(IN := #DWORD_1, N := #statSensorParameter.FineResolutionXist2));
	            IF #statMotionType = 0 THEN
	                //linear axis
	                #statResolutionAbs := #tempIncResolution / #statLeadScrew;
	            ELSE
	                // rotatory axis
	                #statResolutionAbs := #tempIncResolution / 360.0;
	            END_IF;
	            
	        END_IF;
	        IF #statInverseDirection THEN
	            #statResolutionCycl := - #statResolutionCycl;
	            #statResolutionAbs := - #statResolutionAbs;
	        END_IF;
	        
	        #statOldPos := #position;
	        #statIncPos := 0;
	        #statDIncPos := 0.0;
	        #statInitDone := TRUE;
	    END_IF;
	END_IF;
	#statInitOld := #init;
	//  Calculate the position difference
	IF #statModulo.Enable THEN
	    #tempDPos := "LSimaHydTO_GetModuloDifference"(actualValue := #position,
	                                                  oldValue := #statOldPos,
	                                                  startValue := #statModulo.StartValue,
	                                                  length := #statModulo.Length);
	ELSE
	    #tempDPos := #position - #statOldPos;
	END_IF;
	
	#statDIncPos := #statDIncPos + #tempDPos * #statResolutionCycl;
	#tempDIncPosInt := TRUNC_DINT(#statDIncPos);
	#statDIncPos := #statDIncPos - #tempDIncPosInt;
	// only consider the changes
	#statIncPos := #statIncPos + #tempDIncPosInt;
	#tel81in.G1_XIST1 := DINT_TO_DWORD(#statIncPos);
	#statOldPos := #position;
	
	
	// Error acknowledgement
	IF #statError THEN
	    IF #tel81out.G1_STW.AcknowledgeError THEN        // Acknowledge
	        #tel81in.G1_XIST2 := 0;
	        #tel81in.G1_ZSW.SensorError := FALSE;
	        #statError := FALSE;
	    END_IF;
	END_IF;
	
	// interprete the encoder control word  G1_STW
	#tempReqCmd := #tel81out.G1_STW.Command0Request OR #tel81out.G1_STW.Command1Request
	OR #tel81out.G1_STW.Command2Request OR #tel81out.G1_STW.RequestParkingEncoder;
	
	
	IF #tempReqCmd THEN                    // any unsupported comands requested? ==> Error
	    #tel81in.G1_ZSW.SensorError := TRUE;
	    #tel81in.G1_XIST2 := 16#0F01;
	    #statError := TRUE;
	ELSE
	    
	    IF #tel81out.G1_STW.AbsoluteValueCyclically THEN        // request absolute value
	        #tel81in.G1_XIST2 := DINT_TO_DWORD(TRUNC_DINT(#position * #statResolutionAbs));
	        #tel81in.G1_ZSW.AbsoluteValueCyclicallyExecuted := TRUE;
	    ELSE
	        #tel81in.G1_ZSW.AbsoluteValueCyclicallyExecuted := FALSE;
	        #tel81in.G1_XIST2 := 0;
	    END_IF;
	    
	END_IF;
	
	
	
END_FUNCTION_BLOCK

FUNCTION "LSimaHydTO_GetExternalEncoderData" : Void
{ S7_Optimized_Access := 'TRUE' }
AUTHOR : APC_ERLF
FAMILY : LSimaHydTO
VERSION : 1.0
   VAR_INPUT 
      axis {InstructionName := 'TO_ExternalEncoder'; LibVersion := '4.0'} : TO_ExternalEncoder;
   END_VAR

   VAR_OUTPUT 
      inverseDirection : Bool;
      sensorSystem : DInt;
      motionType : DInt;
      leadScrew : LReal;
      modulo {InstructionName := 'TO_Struct_Modulo'; LibVersion := '4.0'} : TO_Struct_Modulo;
      sensorParameter {InstructionName := 'TO_Struct_SensorParameter'; LibVersion := '4.0'} : TO_Struct_SensorParameter;
   END_VAR


BEGIN
	//================================================================================
	//SIEMENS AG // (c)Copyright 2019 All Rights Reserved
	//--------------------------------------------------------------------------------
	//Library:       LSimaHydTO
	//Tested with:   S7-15xx
	//Engineering:   TIA Portal  V15
	//Restrictions:  -
	//Requirements:  S7-1500 (FW 2.5)
	//Functionality: read external encoder parameter  
	//
	//--------------------------------------------------------------------------------
	//Change log table:
	//
	//Version     Date          Expert in charge    Changes applied
	//01.00.00    27.06.2019    APC_ERLF            First released version
	//================================================================================
	
	#inverseDirection := #axis.Sensor.InverseDirection;
	#sensorSystem := #axis.Sensor.System;
	#motionType := #axis.Properties.MotionType;
	#leadScrew := #axis.Mechanics.LeadScrew;
	#modulo.Enable := #axis.Modulo.Enable;
	#modulo.Length := #axis.Modulo.Length;
	#modulo.StartValue := #axis.Modulo.StartValue;
	
	#sensorParameter.DeterminableRevolutions := #axis.Sensor.Parameter.DeterminableRevolutions;
	#sensorParameter.DistancePerRevolution := #axis.Sensor.Parameter.DistancePerRevolution;
	#sensorParameter.FineResolutionXist1 := #axis.Sensor.Parameter.FineResolutionXist1;
	#sensorParameter.FineResolutionXist2 := #axis.Sensor.Parameter.FineResolutionXist2;
	#sensorParameter.Resolution := #axis.Sensor.Parameter.Resolution;
	#sensorParameter.StepsPerRevolution := #axis.Sensor.Parameter.StepsPerRevolution;
	
	
	
END_FUNCTION

FUNCTION "LSimaHydTO_GetPosAxisEncoderData" : Word
{ S7_Optimized_Access := 'TRUE' }
AUTHOR : APC_ERLF
FAMILY : LSimaHydTO
VERSION : 1.0
   VAR_INPUT 
      axis {InstructionName := 'TO_PositioningAxis'; LibVersion := '4.0'} : TO_PositioningAxis;
   END_VAR

   VAR_OUTPUT 
      inverseDirection : Bool;
      sensorSystem : DInt;
      motionType : DInt;
      leadScrew : LReal;
      modulo {InstructionName := 'TO_Struct_Modulo'; LibVersion := '4.0'} : TO_Struct_Modulo;
      sensorParameter {InstructionName := 'TO_Struct_SensorParameter'; LibVersion := '4.0'} : TO_Struct_SensorParameter;
   END_VAR

   VAR_TEMP 
      tempActiveEncoder : Int;
   END_VAR

   VAR CONSTANT 
      MAX_SENSOR_NUMBER : Int := 4;
      ERR_NO_ENCODER_ACTIVE : Word := 16#8200;
   END_VAR


BEGIN
	//================================================================================
	//SIEMENS AG // (c)Copyright 2019 All Rights Reserved
	//--------------------------------------------------------------------------------
	//Library:       LSimaHydTO
	//Tested with:   S7-15xx
	//Engineering:   TIA Portal  V15
	//Restrictions:  -
	//Requirements:  S7-1500 (FW 2.5)
	//Functionality: read pos axis encoder parameter  
	//
	//--------------------------------------------------------------------------------
	//Change log table:
	//
	//Version     Date          Expert in charge    Changes applied
	//01.00.00    27.06.2019    APC_ERLF            First released version
	//================================================================================
	
	FOR #tempActiveEncoder := 1 TO #MAX_SENSOR_NUMBER DO
	  IF #axis.StatusSensor[#tempActiveEncoder].Control THEN
	    EXIT;
	  END_IF;
	END_FOR;
	
	IF #tempActiveEncoder >= 1 AND #tempActiveEncoder <= #MAX_SENSOR_NUMBER THEN
	  #LSimaHydTO_GetPosAxisEncoderData := 0;
	  
	  #inverseDirection := #axis.Sensor[#tempActiveEncoder].InverseDirection;
	  #sensorSystem := #axis.Sensor[#tempActiveEncoder].System;
	  #motionType := #axis.Properties.MotionType;
	  #leadScrew := #axis.Mechanics.LeadScrew;
	  #modulo.Enable := #axis.Modulo.Enable;
	  #modulo.Length := #axis.Modulo.Length;
	  #modulo.StartValue := #axis.Modulo.StartValue;
	  
	  #sensorParameter.DeterminableRevolutions := #axis.Sensor[#tempActiveEncoder].Parameter.DeterminableRevolutions;
	  #sensorParameter.DistancePerRevolution := #axis.Sensor[#tempActiveEncoder].Parameter.DistancePerRevolution;
	  #sensorParameter.FineResolutionXist1 := #axis.Sensor[#tempActiveEncoder].Parameter.FineResolutionXist1;
	  #sensorParameter.FineResolutionXist2 := #axis.Sensor[#tempActiveEncoder].Parameter.FineResolutionXist2;
	  #sensorParameter.Resolution := #axis.Sensor[#tempActiveEncoder].Parameter.Resolution;
	  #sensorParameter.StepsPerRevolution := #axis.Sensor[#tempActiveEncoder].Parameter.StepsPerRevolution;
	  
	ELSE
	  #LSimaHydTO_GetPosAxisEncoderData := #ERR_NO_ENCODER_ACTIVE;
	END_IF;
	
	
	
END_FUNCTION

FUNCTION "LSimaHydTO_GetSyncAxisEncoderData" : Word
{ S7_Optimized_Access := 'TRUE' }
AUTHOR : APC_ERLF
FAMILY : LSimaHydTO
VERSION : 1.0
   VAR_INPUT 
      axis {InstructionName := 'TO_SynchronousAxis'; LibVersion := '4.0'} : TO_SynchronousAxis;
   END_VAR

   VAR_OUTPUT 
      inverseDirection : Bool;
      sensorSystem : DInt;
      motionType : DInt;
      leadScrew : LReal;
      modulo {InstructionName := 'TO_Struct_Modulo'; LibVersion := '4.0'} : TO_Struct_Modulo;
      sensorParameter {InstructionName := 'TO_Struct_SensorParameter'; LibVersion := '4.0'} : TO_Struct_SensorParameter;
   END_VAR

   VAR_TEMP 
      tempActiveEncoder : Int;
   END_VAR

   VAR CONSTANT 
      MAX_SENSOR_NUMBER : Int := 4;
      ERR_NO_ENCODER_ACTIVE : Word := 16#8200;
   END_VAR


BEGIN
	//================================================================================
	//SIEMENS AG // (c)Copyright 2019 All Rights Reserved
	//--------------------------------------------------------------------------------
	//Library:       LSimaHydTO
	//Tested with:   S7-15xx
	//Engineering:   TIA Portal  V15
	//Restrictions:  -
	//Requirements:  S7-1500 (FW 2.5)
	//Functionality: read sync axis encoder parameter  
	//
	//--------------------------------------------------------------------------------
	//Change log table:
	//
	//Version     Date          Expert in charge    Changes applied
	//01.00.00    27.06.2019    APC_ERLF            First released version
	//================================================================================
	
	FOR #tempActiveEncoder := 1 TO #MAX_SENSOR_NUMBER DO
	  IF #axis.StatusSensor[#tempActiveEncoder].Control THEN
	    EXIT;
	  END_IF;
	END_FOR;
	
	IF #tempActiveEncoder >= 1 AND #tempActiveEncoder <= #MAX_SENSOR_NUMBER THEN
	  #LSimaHydTO_GetSyncAxisEncoderData := 0;
	  
	  #inverseDirection := #axis.Sensor[#tempActiveEncoder].InverseDirection;
	  #sensorSystem := #axis.Sensor[#tempActiveEncoder].System;
	  #motionType := #axis.Properties.MotionType;
	  #leadScrew := #axis.Mechanics.LeadScrew;
	  #modulo.Enable := #axis.Modulo.Enable;
	  #modulo.Length := #axis.Modulo.Length;
	  #modulo.StartValue := #axis.Modulo.StartValue;
	  
	  #sensorParameter.DeterminableRevolutions := #axis.Sensor[#tempActiveEncoder].Parameter.DeterminableRevolutions;
	  #sensorParameter.DistancePerRevolution := #axis.Sensor[#tempActiveEncoder].Parameter.DistancePerRevolution;
	  #sensorParameter.FineResolutionXist1 := #axis.Sensor[#tempActiveEncoder].Parameter.FineResolutionXist1;
	  #sensorParameter.FineResolutionXist2 := #axis.Sensor[#tempActiveEncoder].Parameter.FineResolutionXist2;
	  #sensorParameter.Resolution := #axis.Sensor[#tempActiveEncoder].Parameter.Resolution;
	  #sensorParameter.StepsPerRevolution := #axis.Sensor[#tempActiveEncoder].Parameter.StepsPerRevolution;
	ELSE
	  #LSimaHydTO_GetSyncAxisEncoderData := #ERR_NO_ENCODER_ACTIVE;
	END_IF;
	
	
	
END_FUNCTION

FUNCTION "LSimaHydTO_GetModuloDifference" : LReal
{ S7_Optimized_Access := 'TRUE' }
AUTHOR : APC_ERLF
FAMILY : LSimaHydTO
VERSION : 1.0
   VAR_INPUT 
      actualValue : LReal;
      oldValue : LReal;
      startValue : LReal;
      length : LReal;
   END_VAR

   VAR_TEMP 
      tempDifValue : LReal;
   END_VAR


BEGIN
	//================================================================================
	//SIEMENS AG // (c)Copyright 2019 All Rights Reserved
	//--------------------------------------------------------------------------------
	//Library:       LSimaHydTO
	//Tested with:   S7-15xx
	//Engineering:   TIA Portal  V15
	//Restrictions:  -
	//Requirements:  S7-1500 (FW 2.5)
	//Functionality: -   
	//
	//--------------------------------------------------------------------------------
	//Change log table:
	//
	//Version     Date          Expert in charge    Changes applied
	//01.00.00    15.03.2018    APC_ERLF            First released version
	//================================================================================
	
	
	#tempDifValue := #actualValue - #oldValue;
	IF ABS(#tempDifValue) <= #length / 2.0 THEN
	  #LSimaHydTO_GetModuloDifference := #tempDifValue;
	ELSIF #actualValue < #oldValue THEN
	  #LSimaHydTO_GetModuloDifference := #length + #tempDifValue;
	ELSE
	  #LSimaHydTO_GetModuloDifference := - #length + #tempDifValue;
	END_IF;
	
END_FUNCTION

FUNCTION "LSimaHydTO_GetPosAxisCorrection" : LReal
{ S7_Optimized_Access := 'TRUE' }
AUTHOR : APC_ERLF
FAMILY : LSimaHydTO
VERSION : 1.0
   VAR_INPUT 
      axis {InstructionName := 'TO_PositioningAxis'; LibVersion := '4.0'} : TO_PositioningAxis;
   END_VAR

   VAR_OUTPUT 
      accelFactor : LReal;
   END_VAR


BEGIN
	//================================================================================
	//SIEMENS AG // (c)Copyright 2019 All Rights Reserved
	//--------------------------------------------------------------------------------
	//Library:       LSimaHydTO
	//Tested with:   S7-15xx
	//Engineering:   TIA Portal  V15
	//Restrictions:  -
	//Requirements:  S7-1500 (FW 2.5)
	//Functionality: - for internal use
	//
	//--------------------------------------------------------------------------------
	//Change log table:
	//
	//Version     Date          Expert in charge    Changes applied
	//01.00.00    24.04.2020    APC_ERLF            First released version
	//================================================================================
	//
	
	#LSimaHydTO_GetPosAxisCorrection := "LSimaHydTO_GetUnitsCorrection"(lengthUnit:=#axis.Units.LengthUnit,
	                                velocityUnit:=#axis.Units.VelocityUnit,
	                                accelFactor=>#accelFactor);
	
END_FUNCTION

FUNCTION "LSimaHydTO_GetSyncAxisCorrection" : LReal
{ S7_Optimized_Access := 'TRUE' }
AUTHOR : APC_ERLF
FAMILY : LSimaHydTO
VERSION : 1.0
   VAR_INPUT 
      axis {InstructionName := 'TO_SynchronousAxis'; LibVersion := '4.0'} : TO_SynchronousAxis;
   END_VAR

   VAR_OUTPUT 
      accelFactor : LReal;
   END_VAR


